// 	 FOR index := 1 TO GVL.gc_NumberStations DO
// 			GVL.g_Stations[index].P_eProcessMode := E_ProcessMode.Production;		   
// 	   END_FOR
// 		
// 	 
// 
// 	nExecutingSequence := nExecutingSequence +10;
// 
// 	10:
// 	  
// 	   
//   IF fbXPlanarMover[nTestID].P_Enable.Done THEN 
// 		stMoveOnTrackOptions.gap := 120;
// 		stMoveOnTrackOptions.direction := MC_DIRECTION.mcDirectionShortestWay;
// 		stMoveOnTrackOptions.dynamicMode := MC_DYNAMICS_REDUCTION_MODE.AccelerationLimitedVelocity;
// 
// 					
// 				fTargetPosOnTrack[1]:= GVL.g_Tracks[9].P_TrackLength;			
// 				fbXPlanarMover[nTestID].MoveOnTrackExt('move on track', GVL.g_Tracks[9].std, fTargetPosOnTrack[1],
// 								500, 2500, 50000, stMoveOnTrackOptions);
// 		nExecutingSequence := nExecutingSequence +1;
// 		 
// 	END_IF
// 
// 	11:
// 		bMoversInPos := TRUE;
// 		bMoverError := FALSE;
// 		
// 		
// 			bMoversInPos := bMoversInPos AND fbXPlanarMover[nTestID].P_MoveOnTrackExt.Done;
// 			bMoverError := bMoverError OR fbXPlanarMover[nTestID].P_MoveOnTrackExt.Error;
// 	
// 		
// 		IF bMoversInPos THEN
// 			nExecutingSequence := nExecutingSequence + 9;
// 		ELSIF bMoverError THEN
// 			nExecutingSequence := nExecutingSequence +  4;
// 		END_IF
// 
// 	20:
// 		FOR nForCounter:=1 TO GVL.gc_NumberStations DO
// 		IF GVL.g_Stations[nForCounter] <> 0 THEN
// 			GVL.g_Stations[nForCounter].Process();
// 			
// 			IF GVL.g_Stations[nForCounter].P_nErrorCode > 0 THEN
// 				nProcessFeedback := GVL.g_Stations[nForCounter].P_nErrorCode;
// 			END_IF
// 		END_IF
// 	END_FOR	
// 		nExecutingSequence := nExecutingSequence +10;
// 		
// 	30:
// 		stMoveOnTrackOptions.gap := 120;
// 		stMoveOnTrackOptions.direction := MC_DIRECTION.mcDirectionShortestWay;
// 		stMoveOnTrackOptions.dynamicMode := MC_DYNAMICS_REDUCTION_MODE.AccelerationLimitedVelocity;
// 		
// 		fTargetPosOnTrack[1] := GVL.g_Tracks[7].P_TrackLength;;
// 		fbXPlanarMover[nTestID].MoveOnTrackExt('move on track', GVL.g_Tracks[7].std, fTargetPosOnTrack[1],
// 												500, 2500, 50000, stMoveOnTrackOptions
// 		);
// 		nExecutingSequence := nExecutingSequence +1;
// 	31:
// 		// Movers moving on track
// 			bMoversInPos := TRUE;
// 			bMoverError := FALSE;
// 		
// 					bMoversInPos := bMoversInPos AND	fbXPlanarMover[nTestID].P_MoveOnTrackExt.Done;
// 					bMoverError := bMoverError OR fbXPlanarMover[nTestID].P_MoveOnTrackExt.Error;
// 	
// 			IF bMoversInPos THEN
// 			nExecutingSequence := nExecutingSequence + 9;
// 			ELSIF bMoverError THEN
// 			nExecutingSequence := nExecutingSequence + 4;
// 			END_IF
// 
// 
// 	40: 
// 
// 		stMoveOnTrackOptions.gap := 120;
// 		stMoveOnTrackOptions.direction := MC_DIRECTION.mcDirectionShortestWay;
// 		stMoveOnTrackOptions.dynamicMode := MC_DYNAMICS_REDUCTION_MODE.AccelerationLimitedVelocity;
// 		
// 		fTargetPosOnTrack[1] := GVL.g_Tracks[8].P_TrackLength;;
// 		fbXPlanarMover[nTestID].MoveOnTrackExt('move on track', GVL.g_Tracks[8].std, fTargetPosOnTrack[1],
// 												500, 2500, 50000, stMoveOnTrackOptions	);									
// 												
// 												
// 		nExecutingSequence := nExecutingSequence +1;
// 	41:
// 		// Movers moving on track
// 			bMoversInPos := TRUE;
// 			bMoverError := FALSE;
// 		
// 					bMoversInPos := bMoversInPos AND	fbXPlanarMover[nTestID].P_MoveOnTrackExt.Done;
// 					bMoverError := bMoverError OR fbXPlanarMover[nTestID].P_MoveOnTrackExt.Error;
// 	
// 			IF bMoversInPos THEN
// 			nExecutingSequence := nExecutingSequence + 9;
// 			ELSIF bMoverError THEN
// 			nExecutingSequence := nExecutingSequence + 4;
// 			END_IF
// 	
// 	
// 
// 	50:
// 		Execute := FALSE; // must be aborted manually
// 		nExecutingSequence := 0; // endless loop
	
END_CASE
END_METHOD

METHOD MoverPreparation : BOOL
VAR_INPUT
	bReset 	: BOOL;
END_VAR


VAR_INST
	
	nStatePreparation		: DINT;
	
	
	operationMode				: XPlanarOperationMode; 
	
	idx2						: UDINT;

	nTileDcLinkVoltage			: LREAL;
	bTilePowerOK				: BOOL;
	bTilePowerOverview			: ARRAY[1..GVL.gc_MaxNumberTiles] OF BOOL;
	bPowerOK					: BOOL;
	bPowerMissing				: BOOL;
	nTileCount					: UDINT;
	nTileToCheck				: UINT;
	bWithBumperID				: BOOL;	
	nMoverAccessoryIdCount		: ARRAY[1..GVL.gc_nMaxNumberMovers] OF UDINT;	
	
	stStartCheck 				: ST_CheckStartConditionFeedback;
	nLimitExceeded_MoverID		: UDINT;
	bLimitExceeded_Angle 		: BOOL;
	bLimitExceeded_PositionX 	: BOOL;
	bLimitExceeded_PositionY 	: BOOL;	
	fCurrentAngleDeviation		: LREAL;
	fCurrentPositionDeviationX	: LREAL;
	fCurrentPositionDeviationY	: LREAL;	

	sTextTemp					: STRING;

	eMoverAccessoryID			: MoverAccessoryID;

	
	moverCoordComStatus			: CoordinatedMoverCommStatus;
	moverComStatus				: MoverCommunicationStatus;
	
	bMoverCommunicationProblem  : ARRAY[1..GVL.gc_nMaxNumberMovers] OF BOOL;
	bCommunicationProblem		: BOOL;
	
	nMoverToCorrect				: UDINT;
	fMoverOrientationRead		: LREAL;
	fMoverOrientationCorrect	: LREAL;
	bDoRotationCorrection		: BOOL;
	CorrectionPos				: PositionXYC;
	
	bDeterminedMoverID				: BOOL;
	bDerterminedMoverOrientation 	: BOOL;
	
	fPosX							: LREAL;
	fPosY							: LREAL;
	fPosC							: LREAL;
	
	nCommunicationRetryCounter		: UINT;
	
	nMoverToCheck					: UINT;
	
	nMoverID_ErrorCode				: DWORD;
	
	MoverType						: XPlanarMoverType;
	bMoverCanDeterminOrientation	: BOOL;
	
			// Helper
	bDone 					: BOOL;
	idx						: UDINT;
	nForCounter 			: UDINT;	
	nErrorID				: UDINT;
	bMoverError				: BOOL;	
END_VAR
VAR
	sBtn: STRING(13);
END_VAR
IF bReset THEN
	nStatePreparation := 0;
	MoverPreparation := TRUE;
END_IF


	CASE nStatePreparation OF
		
	0:  nStatePreparation := 10;
	

	10: // 1st: Check if the system is in simulation mode or not
		// Simulation > OperationMode = 1
		//     Normal > OperationMode = 0
	    operationMode := fbXPlanarSystem.ipDriver.TcIoXpu(1).GetOperationMode();	
		IF operationMode = 0 THEN
			bPowerMissing := FALSE;
			nStatePreparation := nStatePreparation + 10;
		ELSE
			nStatePreparation := 500;
		END_IF
	
		
	20: // 2nd: Check power of each tile
		(*IF NOT bPowerMissing THEN
			ipVisuMessage.SetInfoMessage('Checking tile power', 'MoverPreparation', nStatePreparation);
		ELSE
			ipVisuMessage.SetErrorMessage('Tile power missing!', 'MoverPreparation', nStatePreparation, 0);	
		END_IF*)
		
		    bPowerOK := TRUE;
		nTileToCheck := 0;
		  nTileCount := fbXPlanarSystem.ipDriver.TcIoXpu(1).GetTileCount();
		
		nStatePreparation := nStatePreparation + 1;
		
	21:
		nTileToCheck := nTileToCheck +1;
		IF nTileToCheck <= nTileCount THEN
			nStatePreparation := nStatePreparation + 1;
		ELSE
			IF bPowerOK THEN
				nStatePreparation := nStatePreparation + 9;
			ELSE
				bPowerMissing := TRUE;
				nStatePreparation := nStatePreparation - 1;
			END_IF
		END_IF
		
	22:
		nTileDcLinkVoltage := fbXPlanarSystem.ipDriver.TcIoXpu(1).TcIoTile(1,nTileToCheck).GetDcLinkVoltage(); 
		IF nTileDcLinkVoltage > 6.0 THEN
			bTilePowerOK := TRUE;
		ELSE
			bTilePowerOK := FALSE;	
		END_IF
		bPowerOK := bPowerOK AND bTilePowerOK;
		bTilePowerOverview[nTileToCheck] := bPowerOK;
		nStatePreparation := nStatePreparation - 1;
		
		
		
	30:// 3rd: Mover re-detection, in case a mover was removed inbetween
	
		// Check if a mover has been lost...
		IF fbXPlanarSystem.CheckValidMovers() THEN
			//ipVisuMessage.SetInfoMessage('Mover re-detection', 'MoverPreparation', nStatePreparation);
		
		nStatePreparation := nStatePreparation + 1;
		END_IF
	
	31:
		IF fbXPlanarSystem.P_CheckValidMovers.bDone THEN
			IF fbXPlanarSystem.P_CheckValidMovers.bMoverLost THEN
				         bDeterminedMoverID := FALSE;
				bDerterminedMoverOrientation := FALSE;
				nStatePreparation := nStatePreparation + 1;
			ELSE
				nStatePreparation := nStatePreparation + 9;
			END_IF
		END_IF
				
		bDeterminedMoverID := FALSE;
		bDerterminedMoverOrientation := FALSE;		
		
		
	32: // Starting mover re-detection
		IF fbXPlanarSystem.UtilityCheckForError(bAutoReset := TRUE) > 0 THEN
			IF fbXPlanarSystem.ipDriver.TcIoXpu(1).SetStartMoverRedetection() THEN	
				nStatePreparation := nStatePreparation +1;
			END_IF
		END_IF
	
	33: // Checking if all movers have been found on the XPlanar surface
		stMoverDetectionInfos := fbXPlanarSystem.ipDriver.TcIoXpu(1).GetMoverDetectionInfos();
		gvl.g_nMoverCount := stMoverDetectionInfos.APM4220Detected ;
		
		
		IF stMoverDetectionInfos.APM4220Detected = stMoverDetectionInfos.APM4220Expected THEN
			nStatePreparation := nStatePreparation +7;
		ELSE
			sTextTemp := 'Mover Missing!  Expected:';
			sTextTemp := CONCAT(sTextTemp, UDINT_TO_STRING(stMoverDetectionInfos.APM4220Expected));
			sTextTemp := CONCAT(sTextTemp, '  Detected:');
			sTextTemp := CONCAT(sTextTemp, UDINT_TO_STRING(stMoverDetectionInfos.APM4220Detected));
			
			//ipVisuMessage.SetErrorMessage(sTextTemp, 'MoverPreparation', nStatePreparation, 0);	
		END_IF
	
	
	 40: // 4th: Checking the position of each mover before enabeling
	 	//ipVisuMessage.SetInfoMessage('Check mover position', 'MoverPreparation', nStatePreparation);
		stMoverDetectionInfos := fbXPlanarSystem.ipDriver.TcIoXpu(1).GetMoverDetectionInfos();	 	
		gvl.g_nMoverCount := stMoverDetectionInfos.APM4220Detected ;
		
		bDone := TRUE;
		FOR idx:=1 TO GVL.g_nMoverCount DO
			stStartCheck := GVL.g_Movers[idx].std.CheckStartConditions();
			IF NOT stStartCheck.bPositionOK THEN
				bDone := FALSE;
				EXIT;
			END_IF			
		END_FOR
	
		IF bDone THEN
			nStatePreparation := nStatePreparation + 2;
		ELSE
			nStatePreparation := nStatePreparation + 1;
		END_IF
			
	 41: // Position-Check failed:
		 // Except for rotation-points between four quadrants the angle limit of the c-axis is +/- 10.0°
		 // At rotation-points the max position deviation is +/-1mm in x/y-direction  	
				nLimitExceeded_MoverID := stStartCheck.nMoverID;
				  bLimitExceeded_Angle := stStartCheck.bAngleLimitExceeded;
			  bLimitExceeded_PositionX := stStartCheck.bPositionXLimitExceeded;
			  bLimitExceeded_PositionY := stStartCheck.bPositionYLimitExceeded;	
				fCurrentAngleDeviation := stStartCheck.fCurrentAngleDeviation;
			fCurrentPositionDeviationX := stStartCheck.fCurrentPositionDeviationX;
			fCurrentPositionDeviationY := stStartCheck.fCurrentPositionDeviationY;
	
			sTextTemp := 'Position Check Failed! - Mover ';
			sTextTemp := CONCAT(sTextTemp, UDINT_TO_STRING(nLimitExceeded_MoverID));
			sTextTemp := CONCAT(sTextTemp, ' too far away from rotation point.');
			
			//ipVisuMessage.SetErrorMessage(sTextTemp, 'MoverPreparation', nStatePreparation, 0);	
			
			nStatePreparation := nStatePreparation - 1;
			
	42:		//ipVisuMessage.ClearAllMessages();
			nStatePreparation := nStatePreparation + 8;
		
		
		
	50: // 5th: Check if movers with accessory MoverID are present. If yes, do mover identification before enabeling all movers.	
		bWithBumperID := FALSE;
			
		IF fbXPlanarSystem.UtilityCheckForError(bAutoReset := TRUE) > 0 THEN
			FOR idx:=1 TO GVL.g_nMoverCount DO
				nMoverAccessoryIdCount[idx] := fbXPlanarSystem.ipDriver.TcIoXpu(1).TcIoMover(UDINT_TO_UINT(idx)).GetMoverAccessoryIdCount();
			END_FOR
			
			FOR idx:=1 TO GVL.g_nMoverCount DO
				FOR idx2:=1 TO nMoverAccessoryIdCount[idx] DO
					eMoverAccessoryID := fbXPlanarSystem.ipDriver.TcIoXpu(1).TcIoMover(UDINT_TO_UINT(idx)).GetMoverAccessoryID(UDINT_TO_INT(idx2));
					
					IF eMoverAccessoryID = MoverAccessoryID.APM9001_0000 THEN
						// Note: With the current driver release (3.2209.36.0) mover identification only works if all movers are equiped with ID bumpers!
						bWithBumperID := TRUE;						
					END_IF
				END_FOR
			END_FOR
		END_IF

			
		IF bWithBumperID THEN
			nStatePreparation := nStatePreparation + 10;
		ELSE
			nStatePreparation := 500;
		END_IF
		
	
	60: // 6th: Do mover identification
		//ipVisuMessage.SetInfoMessage('Start mover-identification', 'MoverPreparation', nStatePreparation);
	
		IF NOT bDeterminedMoverID THEN
			IF fbXPlanarSystem.UtilityCheckForError(bAutoReset := TRUE) > 0 THEN
// 				IF fbXPlanarSystem.ipDriver.TcIoXpu(1).SetCoordMoverCommunicationCmd(CoordinatedMoverCommCommand.IdentifyAndAssignPossible) THEN
				IF fbXPlanarSystem.ipDriver.TcIoXpu(1).SetCoordMoverCommunicationCmd(CoordinatedMoverCommCommand.IdentifyBTNsAndRearrangeMovers) THEN
					nStatePreparation := nStatePreparation +1;
				END_IF	
			END_IF
		ELSE
			nStatePreparation := nStatePreparation +10;
		END_IF
	
	61:
		IF fbXPlanarSystem.UtilityCheckForError(bAutoReset := TRUE) > 0 THEN			
			moverCoordComStatus := fbXPlanarSystem.ipDriver.TcIoXpu(1).GetCoordMoverCommStatus();
			
			IF moverCoordComStatus = CoordinatedMoverCommStatus.CommunicationSuccessful THEN
				bDeterminedMoverID := TRUE;
				//ipVisuMessage.ClearAllMessages();
				nStatePreparation := nStatePreparation + 4;
			ELSIF moverCoordComStatus = CoordinatedMoverCommStatus.CommunicationFailed THEN
				nStatePreparation := nStatePreparation + 1;	
			END_IF
			
		END_IF
		
	62:	IF fbXPlanarSystem.UtilityCheckForError(bAutoReset := TRUE) > 0 THEN	
			nMoverID_ErrorCode := fbXPlanarSystem.ipDriver.TcIoXpu(1).GetCoordMoverCommunicationErrorId();
			//ipVisuMessage.SetErrorMessage('Mover Identification Failed!', 'MoverPreparation', nStatePreparation, nMoverID_ErrorCode);
		END_IF
		
		//IF ipVisuMessage.CheckAknowledge()  THEN
		nStatePreparation := 0;	
		//END_IF
	
	65: 
		FOR idx:=1 TO GVL.g_nMoverCount DO
			fbMover[idx].P_MoverID := fbXPlanarSystem.ipDriver.TcIoXpu(1).TcIoMover(UDINT_TO_UINT(idx)).GetIdentifiedMoverBtn();
		END_FOR
		nStatePreparation := nStatePreparation + 5;
	70: // 7th: Determine Mover-Orientation
	
		// Note: At the time of creation of this example code only APM4330 was able to determine its orientation.
		//       Change the code according to newer driver releases and availability of the orientation feature.
		bMoverCanDeterminOrientation := TRUE;
		FOR idx:=1 TO GVL.g_nMoverCount DO
			MoverType := fbXPlanarSystem.ipDriver.TcIoXpu(1).TcIoMover(UDINT_TO_UINT(idx)).GetMoverType();
			IF MoverType <> XPlanarMoverType.APM4330 THEN
				bMoverCanDeterminOrientation := FALSE;
			END_IF
		END_FOR
			
		IF bMoverCanDeterminOrientation THEN
			IF NOT bDerterminedMoverOrientation THEN
				//ipVisuMessage.SetInfoMessage('Mover orientation determination', 'MoverPreparation', nStatePreparation);
				IF fbXPlanarSystem.UtilityCheckForError(bAutoReset := TRUE) > 0 THEN
					IF fbXPlanarSystem.ipDriver.TcIoXpu(1).SetCoordMoverCommunicationCmd(CoordinatedMoverCommCommand.DetermineOrientations) THEN
						nStatePreparation := nStatePreparation + 1;	
					END_IF
				END_IF
			ELSE
				nStatePreparation := nStatePreparation + 20;		
			END_IF
		ELSE
			nStatePreparation := nStatePreparation + 20;
		END_IF
	
		
	71: // Check if communication is active
		IF fbXPlanarSystem.UtilityCheckForError(bAutoReset := TRUE) > 0 THEN
			moverCoordComStatus := fbXPlanarSystem.ipDriver.TcIoXpu(1).GetCoordMoverCommStatus();
			IF moverCoordComStatus = CoordinatedMoverCommStatus.CommunicationInProcess THEN
				nStatePreparation := nStatePreparation + 1;	
			END_IF
		END_IF
	
		
	72: // Wait for orientation determination finished
		IF fbXPlanarSystem.UtilityCheckForError(bAutoReset := TRUE) > 0 THEN
			moverCoordComStatus := fbXPlanarSystem.ipDriver.TcIoXpu(1).GetCoordMoverCommStatus();
			IF moverCoordComStatus = CoordinatedMoverCommStatus.CommunicationSuccessful THEN
				nStatePreparation := nStatePreparation + 8;	
			ELSIF moverCoordComStatus = CoordinatedMoverCommStatus.CommunicationFailed THEN
				IF nCommunicationRetryCounter <= 5 THEN
					nCommunicationRetryCounter := nCommunicationRetryCounter +1;
					nStatePreparation := nStatePreparation - 2;	
				ELSE
					nStatePreparation := nStatePreparation + 1;	
				END_IF
			END_IF
		END_IF
		
				
	73:	// Check which movers do not communicate correctly:
		nMoverToCheck := 0;
		nStatePreparation := nStatePreparation + 1;
		
	74: nMoverToCheck := nMoverToCheck +1;
		IF nMoverToCheck <= GVL.g_nMoverCount THEN
			IF fbXPlanarSystem.UtilityCheckForError(bAutoReset := TRUE) > 0 THEN
				IF fbXPlanarSystem.ipDriver.TcIoXpu(1).TcIoMover(nMoverToCheck).SetMoverCommunicationCommand(MoverCommunicationCommand.DetermineOrientation) THEN
					nStatePreparation := nStatePreparation + 1;
				END_IF
			END_IF
		ELSE
			FOR idx:=1 TO GVL.g_nMoverCount DO
				bCommunicationProblem := FALSE;
				IF bMoverCommunicationProblem[idx] THEN
					bCommunicationProblem := TRUE;	
				END_IF
			END_FOR
			
			IF bCommunicationProblem THEN
				sTextTemp := 'Mover Communication Problem: ';
				FOR idx:=1 TO GVL.g_nMoverCount DO
					IF bMoverCommunicationProblem[idx] THEN
						sTextTemp := CONCAT(sTextTemp, ' M');
						sTextTemp := CONCAT(sTextTemp, UDINT_TO_STRING(idx));
					END_IF
				END_FOR				
				//ipVisuMessage.SetErrorMessage(sTextTemp, sTextTemp, nStatePreparation, 0);
			ELSE
				nStatePreparation := nStatePreparation - 4;	
			END_IF
		END_IF
		
	75: moverComStatus := fbXPlanarSystem.ipDriver.TcIoXpu(1).TcIoMover(nMoverToCheck).GetCommunicationStatus();
		IF moverComStatus = MoverCommunicationStatus.CommunicationSuccessful THEN
			bMoverCommunicationProblem[nMoverToCheck] := FALSE;
			nStatePreparation := nStatePreparation - 1;
		ELSIF moverComStatus = MoverCommunicationStatus.CommunicationFailed THEN
			bMoverCommunicationProblem[nMoverToCheck] := TRUE;
			nStatePreparation := nStatePreparation - 1;
		END_IF
		
		
	80:	// Rotation-Angle modulo adaption
		//ipVisuMessage.SetInfoMessage('Rotation-Angle modulo adaption', 'MoverPreparation', nStatePreparation);
		nMoverToCorrect := 0;
		nStatePreparation := nStatePreparation + 1;	
		
	81:	nMoverToCorrect := nMoverToCorrect +1;
		IF nMoverToCorrect <= GVL.g_nMoverCount THEN
			fMoverOrientationRead    := GVL.g_Movers[nMoverToCorrect].std.P_ActPosition.c; 
			fMoverOrientationCorrect := fMoverOrientationRead;
			 bDoRotationCorrection := FALSE;
			nStatePreparation := nStatePreparation + 1;	
		ELSE
			bDerterminedMoverOrientation := TRUE;
			nStatePreparation := nStatePreparation + 9;	
		END_IF
		
	82:	IF fMoverOrientationCorrect >= 0 THEN
			IF fMoverOrientationCorrect > 360.0 THEN
				fMoverOrientationCorrect := fMoverOrientationCorrect - 180.0;
				bDoRotationCorrection := TRUE;
			ELSE
				nStatePreparation := nStatePreparation + 1;
			END_IF
		ELSE
			IF fMoverOrientationCorrect < 360.0 THEN
				fMoverOrientationCorrect := fMoverOrientationCorrect + 180.0;
				bDoRotationCorrection := TRUE;
			ELSE
				nStatePreparation := nStatePreparation + 1;
			END_IF
		END_IF			
		
		
	83:	IF bDoRotationCorrection THEN
			
			fPosX := GVL.g_Movers[nMoverToCorrect].std.P_ActPosition.x;
			fPosY := GVL.g_Movers[nMoverToCorrect].std.P_ActPosition.y;
			fPosC := GVL.g_Movers[nMoverToCorrect].std.P_ActPosition.c;
	
			CorrectionPos.SetValuesXYC(fPosX, fPosY, fMoverOrientationCorrect);	
	
			GVL.g_Movers[nMoverToCorrect].std.SetMoverPosition('Correction', CorrectionPos);
			
			nStatePreparation := nStatePreparation + 1;	
		ELSE
			nStatePreparation := nStatePreparation - 2;
		END_IF
		
	84:
		IF GVL.g_Movers[nMoverToCorrect].std.P_SetMoverPosition.Done THEN
			nStatePreparation := nStatePreparation - 3;
		ELSIF GVL.g_Movers[nMoverToCorrect].std.P_SetMoverPosition.Error THEN
			nErrorID := GVL.g_Movers[nMoverToCorrect].std.P_SetMoverPosition.ErrorID;
			//ipVisuMessage.SetErrorMessage('Rotation-Angle modulo adaption', 'MoverPreparation', nStatePreparation, nErrorID);
			GVL.g_Movers[nMoverToCorrect].P_ErrorID := UDINT_TO_INT(nErrorID);
			GVL.g_Movers[nMoverToCorrect].P_Error := TRUE;
		END_IF
		

	90: nStatePreparation := 500;
	
			
	500: // Done
	//	nStatePreparation := 0;
		MoverPreparation := TRUE;		
			
		
	END_CASE


	//ipVisuMessage.StateUpdate(nStatePreparation, 'MoverPreparation');
END_METHOD

METHOD MoverRecovery : BOOL
VAR_INPUT
	bReset : BOOL;
END_VAR

VAR
	index : UDINT;
	ipMoverApplication: INT;
END_VAR

VAR_INST
	
	stOptionsJoinTrack				: ST_JoinTrackOptions;
	bMoversJoined 					: BOOL;
	bMoverError 					: BOOL;
	bMoverOrientationSet			: BOOL;
	bClearStation 					:ARRAY [1..GVL.gc_NumberStations] OF BOOL;
	bStationCleared					:bool;
	nMoverToTurn					: UDINT;
	nMoverToTurnBack				: UDINT;
	nTrackToCheck					:UDINT; 
	nDistanceToTrack				:LREAL;
	nDistanceToTargetTrack			: ARRAY[1..moverCount] OF REAL;
	nTargetTrack					: ARRAY[1..moverCount] OF UDINT;
	
	
	
	fRecoveryRotTarget				: LREAL;
	fRecoveryRotVel					: LREAL :=  360.0;
	fRecoveryRotAcc					: LREAL := 1800.0;
	fRecoveryRotJerk				: LREAL := 9000.0;
	stRotationOptions				: ST_MoveCOptions;




	
END_VAR
IF bReset THEN
	MoverRecovery := FALSE;
	nRecoverySequence := 0;
END_IF

CASE nRecoverySequence OF
	0:
		bMoversJoined := FALSE;
		bMoverError := FALSE;
		nMoverToTurn := 0;
		IF NOT bReset THEN
			nRecoverySequence := nRecoverySequence + 1;
		END_IF
		
	1: 	//set rotary orienation 
	
		FOR index := 1 TO gvl.g_nMoverCount DO
		fbXPlanarMover[index].MoveA('', 0, 100, 1000, 1000, 10000);
		fbXPlanarMover[index].MoveB('', 0, 100, 1000, 1000, 10000);
 		fbXPlanarMover[index].MoveC('', 0, 180, 1800, 1800, 18000, 0);
		
		END_FOR

		nRecoverySequence := nRecoverySequence + 1;
	
	2: 
		bMoverOrientationSet:= TRUE; 
		FOR index := 1 TO  gvl.g_nMoverCount DO
			IF fbXPlanarMover[index].P_MoveA.Done AND fbXPlanarMover[index].P_MoveB.Done AND fbXPlanarMover[index].P_MoveC.Done THEN 
				bMoverOrientationSet:= TRUE; 
			ELSE 
				bMoverOrientationSet:= FALSE; 
				
			END_IF
		END_FOR
		
		IF bMoverOrientationSet THEN
			nRecoverySequence := nRecoverySequence + 8;
	
		END_IF
	
	10:
	
		nMoverToTurn := nMoverToTurn +1;
		IF nMoverToTurn > gvl.g_nMoverCount THEN
				nRecoverySequence := nRecoverySequence +3;
			ELSE
				IF GVL.g_Movers[nMoverToTurn].std.P_IsPresent THEN

					fRecoveryRotTarget 				  := GVL.g_Movers[nMoverToTurn].std.P_ClosestQuaterAngle;	
					stRotationOptions.additionalTurns := 0;
					stRotationOptions.direction		  := Tc3_Mc3PlanarMotion.MC_direction.mcDirectionNonModulo;	
					
					GVL.g_Movers[nMoverToTurn].std.MoveC('Recovery - unfinished rotation', fRecoveryRotTarget, fRecoveryRotVel, fRecoveryRotAcc, fRecoveryRotAcc, fRecoveryRotJerk, stRotationOptions);
					nRecoverySequence := nRecoverySequence +1;				
				END_IF	
			END_IF
		
	
	11:
			IF GVL.g_Movers[nMoverToTurn].std.P_MoveC.Done THEN
				nRecoverySequence := nRecoverySequence -1;	
			ELSIF GVL.g_Movers[nMoverToTurn].std.P_MoveC.Error THEN
				nRecoverySequence := nRecoverySequence +1;	
			END_IF
			
	12: 		// Check error ID and react accordingly
			nErrorID := GVL.g_Movers[nMoverToTurn].std.P_MoveC.ErrorID;
			GVL.g_Movers[nMoverToTurn].P_ErrorID := UDINT_TO_INT(nErrorID);
			GVL.g_Movers[nMoverToTurn].P_Error := TRUE;

			// In case rotation is not possible due to collision with another mover proceed without rotation correction.
			IF nErrorID = 33158 THEN
				nRecoverySequence := nRecoverySequence -2;
			END_IF

	13: 	nRecoverySequence := 100;	

		    
	100: 
			bStationCleared:=TRUE;
			bClearStation[GVL.PuncherStation]:=fbPuncherStation.Clear();
			bClearStation[GVL.PuncherSeparateStation]:=fbPuncherSeparateStation.Clear();
			bClearStation[GVL.PuncherBufferStation]:=fbPuncherBufferStation.Clear();
	
	FOR  index := 1 TO  GVL.gc_NumberStations DO
		IF bClearStation[index] THEN
			bStationCleared:=TRUE;
			ELSE
				bStationCleared:=FALSE;
		END_IF
	END_FOR
	IF bStationCleared THEN
			nRecoverySequence := 200;

		END_IF
		
// 	110: // look for for nearest track 
// 	
// 	
// 	FOR nMoverToTurnBack := 1 TO  gvl.g_nMoverCount DO
// 		nDistanceToTargetTrack[nMoverToTurnBack]:= 999999;
// 		
// 		FOR nTrackToCheck :=1 TO GVL.gc_NumberTracks DO 
// 		nDistanceToTrack := fbXPlanarMover[ nMoverToTurnBack].GetDistanceToTrack(GVL.g_Tracks[nTrackToCheck].std);
// 		
// 		IF nDistanceToTrack < nDistanceToTargetTrack[nMoverToTurnBack] AND nDistanceToTrack<> -1 THEN 
// 			nDistanceToTargetTrack[nMoverToTurnBack]:=nDistanceToTrack;
// 			nTargetTrack[nMoverToTurnBack] :=nTrackToCheck;
// 		END_IF
// 		
// 	END_FOR
// 	
// 	END_FOR
// 	
// 	nRecoverySequence := nRecoverySequence +10;
// 	
// 	120: // join to track
// 
// 		stOptionsJoinTrack.useOrientation := TRUE;
// 		
// 		FOR index := 1 TO gvl.g_nMoverCount DO
// 		IF fbXPlanarMover[index].P_CommandMode<> MC_PLANAR_MOVER_COMMAND_MODE.OnTrack THEN
// 			fbXPlanarMover[index].JoinTrack('Joining track', GVL.g_Tracks[nTargetTrack[index]].std, 250, 1250, 12500, stOptionsJoinTrack);
// 			
// 		END_IF
// 		
// 			
// END_FOR
// 	
// 		nRecoverySequence := nRecoverySequence + 1;
// 		
// 	121:
// 		bMoversJoined := TRUE;
// 		bMoverError := FALSE;
// 		FOR index := 1 TO moverCount DO
// 			bMoversJoined := bMoversJoined AND fbXPlanarMover[index].P_JoinTrack.Done;
// 			IF  fbXPlanarMover[index].P_JoinTrack.Done THEN 
// 				gvl.g_Movers[index].P_TrackId:=nTargetTrack[index];
// 			END_IF
// 			bMoverError := bMoverError OR fbXPlanarMover[index].P_JoinTrack.Error;			
// 		END_FOR
// 		
// 	IF bMoversJoined THEN
// 			nRecoverySequence := nRecoverySequence + 9;
// 	ELSIF bMoverError THEN
//  			nRecoverySequence := nRecoverySequence + 4;
// 	END_IF
// 		
		
// 	130: //send mover to station 
// 	  	  
// 		FOR index := 1 TO gvl.g_nMoverCount DO
// 			 IF fbXPlanarMover[index].P_TrackId= GVL.TrackPuncherWellplate THEN 
// 				 fbPuncherStation.P_List_Switch_Input_W.AddMover(GVL.g_Movers[index].std);
// 		
// 			
// 			 END_IF
// 		END_FOR
// 
// 		nRecoverySequence := 200;

	200: 
		MoverRecovery := TRUE;
		
END_CASE
END_METHOD

METHOD Resetting : BOOL
VAR_INPUT
END_VAR

VAR
	index : UDINT;
	MC_PLANNAR_: ST_CommandReturn;
END_VAR


VAR_INST
	
	nTrackToEnable		: UDINT;
	stProductDataClear 	: ST_ProductData;
	stOptionsJoinTrack				: ST_JoinTrackOptions;
	bMoversJoined 					: BOOL;
	bMoverError 					: BOOL;
	nMoverToTurn					: UDINT;
	nMoverToTurnBack				: UDINT;
	nTrackToCheck					:UDINT; 
	nDistanceToTrack				:LREAL;
	nDistanceToTargetTrack			: ARRAY[1..moverCount] OF REAL;
	nTargetTrack					: ARRAY[1..moverCount] OF UDINT;
	
END_VAR
nErrorID := 0;

CASE nResettingSequence OF 
	
	0: // Enter 
		nResettingSequence := 10;
		
		
		
	10: // Reset all movers
		IF fbXPlanarSystem.ResetMovers() THEN
		//	ipVisuMessage.SetInfoMessage('RESET all movers', 'Resetting', nResettingSequence);
			nResettingSequence := nResettingSequence +1;			
		END_IF
		
	11: IF fbXPlanarSystem.P_ResetMovers.Done THEN
			nResettingSequence := nResettingSequence +9;
		ELSIF fbXPlanarSystem.P_ResetMovers.Error THEN
			nResettingSequence := nResettingSequence +1;	
		END_IF

	12:	// Check error ID and react accordingly
		nErrorID := fbXPlanarSystem.P_EnableMovers.ErrorID;
		//ipVisuMessage.SetErrorMessage('RESET movers failed', 'Resetting', nResettingSequence, nErrorID);					
		
		
		
	20:	// Reset all tracks
		IF fbXPlanarSystem.ResetTracks() THEN
			//ipVisuMessage.SetInfoMessage('RESET all tracks', 'Resetting', nResettingSequence);
			nResettingSequence := nResettingSequence +1;
		END_IF
		
	21: IF fbXPlanarSystem.P_ResetTracks.Done THEN
			nResettingSequence := nResettingSequence +19;
	 	ELSIF fbXPlanarSystem.P_ResetTracks.Error THEN
			nResettingSequence := nResettingSequence +1;	
		END_IF
	
	22:	// Check error ID and react accordingly
		nErrorID := fbXPlanarSystem.P_EnableMovers.ErrorID;
		//ipVisuMessage.SetErrorMessage('RESET tracks failed', 'Resetting', nResettingSequence, nErrorID);			
		
	
		
// 	30:	// Reset MotionSystemApplication
// 		IF ipMotionSystemApplication.Reset() THEN
// 		//	ipVisuMessage.SetInfoMessage('RESET MotionSystemApplication', 'Resetting', nResettingSequence);
// 			nResettingSequence := nResettingSequence +10;
// 		END_IF
	
				
	40:  // Cleaning all process data
		FOR idx:=1 TO GVL.g_nMoverCount DO
		//	ipMoverApplication[idx].P_ProductData := stProductDataClear;
		END_FOR
		nResettingSequence := nResettingSequence+10;
		
	50: // check if any mover is disable 
			
		FOR index := 1 TO gvl.g_nMoverCount DO
			 IF fbXPlanarMover[index].P_State=MC_PLANAR_STATE.Disabled THEN 
				 nResettingSequence := nResettingSequence + 1;
				 RETURN; 
			 END_IF
		END_FOR
			 nResettingSequence :=100;
	 
	51:	// enable movers
			IF fbXPlanarSystem.EnableMovers() THEN
				nResettingSequence := nResettingSequence + 1;
			END_IF
	
	52: // wait for enabling
		IF fbXPlanarSystem.P_EnableMovers.Done THEN
			nResettingSequence := 100;
		ELSIF fbXPlanarSystem.P_EnableMovers.Error THEN
			nResettingSequence := nResettingSequence + 3;
			nErrorID := fbXPlanarSystem.P_EnableMovers.ErrorID;
 		END_IF
		
// 	60:  // look for for nearest track 
// 	
// 		FOR nMoverToTurnBack := 1 TO  gvl.g_nMoverCount DO
// 			nDistanceToTargetTrack[nMoverToTurnBack]:= 999999;
// 			
// 			FOR nTrackToCheck :=1 TO 10 DO//GVL.gc_NumberTracks DO 
// 			nDistanceToTrack := fbXPlanarMover[ nMoverToTurnBack].GetDistanceToTrack(GVL.g_Tracks[nTrackToCheck].std);
// 			
// 				IF nDistanceToTrack < nDistanceToTargetTrack[nMoverToTurnBack] THEN 
// 					nDistanceToTargetTrack[nMoverToTurnBack]:=nDistanceToTrack;
// 					nTargetTrack[nMoverToTurnBack] :=nTrackToCheck;
// 				END_IF
// 			
// 			END_FOR
// 	
// 		END_FOR
// 		
// 	nResettingSequence := nResettingSequence +10;
// 	
// 	70: // join to track
// 
// 		stOptionsJoinTrack.useOrientation := TRUE;
// 		
// 		FOR index := 1 TO gvl.g_nMoverCount DO
// 		IF fbXPlanarMover[index].P_CommandMode<> MC_PLANAR_MOVER_COMMAND_MODE.OnTrack THEN
// 			fbXPlanarMover[index].JoinTrack('Joining track', GVL.g_Tracks[nTargetTrack[index]].std, 250, 1250, 12500, stOptionsJoinTrack);
// 			END_IF
// 
// END_FOR
// 	
// 		nResettingSequence := nResettingSequence + 1;
// 		
// 	71:
// 		bMoversJoined := TRUE;
// 		bMoverError := FALSE;
// 		FOR index := 1 TO moverCount DO
// 			bMoversJoined := bMoversJoined AND fbXPlanarMover[index].P_JoinTrack.Done;
// 			bMoverError := bMoverError OR fbXPlanarMover[index].P_JoinTrack.Error;			
// 		END_FOR
// 		
// 	IF bMoversJoined THEN
// 			nResettingSequence := 100;
// 	ELSIF bMoverError THEN
//  			nResettingSequence := nResettingSequence + 4;
// 	END_IF
// 		
	
	100: // Reset done
		//ipVisuMessage.SetInfoMessage('RESET finished', 'Resetting', 0);
	
		nResettingSequence := 0; 
		         Resetting := TRUE;

END_CASE



//ipVisuMessage.StateUpdate(nResettingSequence, 'Resetting');
END_METHOD

METHOD Starting : BOOL
VAR_INPUT
	bReset : BOOL;
END_VAR

VAR 
	nErrorID : UDINT;
	nMoverIndex: UDINT;
END_VAR
IF bReset THEN
	Starting := FALSE;
	nStartingSequence := 0;
END_IF

CASE nStartingSequence OF
	0: //init
		Execute(bReset := TRUE);
		MoverRecovery(bReset := TRUE);
		IF NOT bReset THEN
			nStartingSequence := nStartingSequence + 10;
		END_IF
	10: // enable collision avoidance group
		IF fbXPlanarSystem.EnableGroup() THEN
			nStartingSequence := nStartingSequence + 1;
		END_IF
	11:
		IF fbXPlanarSystem.P_EnableGroup.Done THEN
			nStartingSequence := nStartingSequence + 9;
		ELSIF fbXPlanarSystem.P_EnableGroup.Error THEN
			nStartingSequence := nStartingSequence + 4;
			nErrorID := fbXPlanarSystem.P_EnableGroup.ErrorID;
		END_IF
	20: // add environment 
		IF fbXPlanarSystem.AddEnvironmentToGroup() THEN
			nStartingSequence := nStartingSequence + 1;
		END_IF
	21: 
		IF fbXPlanarSystem.P_AddEnviromentToGroup.Done THEN
			nStartingSequence := nStartingSequence + 9;
		ELSIF fbXPlanarSystem.P_AddEnviromentToGroup.Error THEN
			nStartingSequence := nStartingSequence + 4;
			nErrorID := fbXPlanarSystem.P_AddEnviromentToGroup.ErrorID;
		END_IF
		
	30:
		IF fbXPlanarSystem.EnableTracks() THEN
			nStartingSequence := nStartingSequence + 1;
		END_IF
	
	31: 
		IF fbXPlanarSystem.P_EnableTracks.Done THEN
			nStartingSequence := nStartingSequence + 9;
		ELSIF fbXPlanarSystem.P_EnableTracks.Error THEN
			nStartingSequence := nStartingSequence + 4;
			nErrorID := fbXPlanarSystem.P_EnableTracks.ErrorID;
		END_IF
	
			
	40:
		IF fbXPlanarSystem.AddTracksToGroup() THEN
			nStartingSequence := nStartingSequence + 1;
		END_IF
	
	41: 
		IF fbXPlanarSystem.P_AddTracksToGroup.Done THEN
			nStartingSequence := nStartingSequence + 1;
		ELSIF fbXPlanarSystem.P_AddTracksToGroup.Error THEN
			nStartingSequence := nStartingSequence + 4;
			nErrorID := fbXPlanarSystem.P_AddTracksToGroup.ErrorID;
		END_IF
		
	42: // Prepare all movers
		IF MoverPreparation(bReset:=TRUE) THEN
			nStartingSequence := nStartingSequence + 1;
		END_IF
		
	43:
		IF MoverPreparation(bReset:=FALSE) THEN
			nStartingSequence := nStartingSequence + 7;
		END_IF	
		
	50: // enable movers
		IF fbXPlanarSystem.EnableMovers() THEN
			nStartingSequence := nStartingSequence + 1;
		END_IF
	51: // wait for enabling
		IF fbXPlanarSystem.P_EnableMovers.Done THEN
			nStartingSequence := nStartingSequence + 9;
		ELSIF fbXPlanarSystem.P_EnableMovers.Error THEN
			nStartingSequence := nStartingSequence + 4;
			nErrorID := fbXPlanarSystem.P_EnableMovers.ErrorID;
		END_IF
	60: // add movers to group
		IF fbXPlanarSystem.AddMoversToGroup() THEN
			nStartingSequence := nStartingSequence + 1;
		END_IF
	61: // wait for enabling
		IF fbXPlanarSystem.P_AddMoversToGroup.Done THEN
			nStartingSequence := nStartingSequence + 1;
		ELSIF fbXPlanarSystem.P_AddMoversToGroup.Error THEN
			nStartingSequence := nStartingSequence + 4;
			nErrorID := fbXPlanarSystem.P_AddMoversToGroup.ErrorID;
		END_IF
	62:
	 	FOR nMoverIndex := 1 TO GVL.g_nMoverCount DO
			GVL.g_Movers[nMoverIndex].std.P_Id := UDINT_TO_UINT(nMoverIndex);
		END_FOR
		nStartingSequence := nStartingSequence + 8;
	70:
		IF MoverRecovery(bReset := FALSE) THEN
			nStartingSequence := nStartingSequence + 10;
		END_IF
	80: 
		Starting := TRUE;
END_CASE
END_METHOD

METHOD Startup : BOOL
VAR_INPUT
	bReset : BOOL;
END_VAR

VAR
	index : UDINT;
		stMoverDetectionInfos   : ST_TcIoMoverDetectionInfos;
		detectedMovers:UDINT;
END_VAR

VAR_INST
	aTrackTable : ARRAY[1..maxTrackCount] OF FB_TrackTable;
	nTrackIdx: UDINT;
	nStationToInit : UINT;
	
	nStartFromTrack : UDINT;
	nEndAtTrack : UDINT;
	bCloseLoop : BOOL;
END_VAR
IF bReset THEN
	Startup := FALSE;
	nStartupSequence := 0;
END_IF

CASE nStartupSequence OF
	0: //init
		bAssignmentComplete := FALSE;
		IF NOT bReset THEN
			nStartupSequence := nStartupSequence + 1;
		END_IF

	1: //assign mover to system
		
		FOR index := 1 TO MoverCount DO
			fbMover[index].std := THIS^.fbXPlanarMover[index];
		END_FOR	
		//nStartupSequence := nStartupSequence + 1;
	
		FOR index := 1 TO moverCount DO
			fbXPlanarSystem.SetMoverStandard(index, THIS^.fbXPlanarMover[index]);
		END_FOR
		
		nStartupSequence := nStartupSequence + 1;
		
	2:  // Movers to global mover interface
		FOR index := 1 TO MoverCount DO
			GVL.g_Movers[index] := THIS^.fbMover[index];
			THIS^.fbMover[index].P_MoverIndex := UDINT_TO_INT(index); 
		END_FOR	
		nStartupSequence := nStartupSequence + 1;
	
	3:  // Assigning global Track-Interfaces
		GVL.g_Tracks[GVL.TrackPuncherWellplate] := THIS^.fbTrackPuncherWellplate;
		GVL.g_Tracks[GVL.TrackBufferPuncher] := THIS^.fbTrackBufferPuncher;
		GVL.g_Tracks[GVL.TrackStradeFirstSeg] := THIS^.fbTrackStradeFirstSeg;
		GVL.g_Tracks[GVL.TrackStradeSecondSeg] := THIS^.fbTrackStradeSecondSeg;
		GVL.g_Tracks[GVL.TrackPipettePreBuffer] := THIS^.fbTrackPipettePreBuffer;
		GVL.g_Tracks[GVL.TrackPipette] := THIS^.fbTrackPipette;
		GVL.g_Tracks[GVL.TrackPipettePostBuffer] := THIS^.fbTrackPipettePostBuffer;
		GVL.g_Tracks[GVL.TrackPipetteBufferCon] := THIS^.fbTrackPipetteBufferCon;
		GVL.g_Tracks[GVL.TrackUserInteraction] := THIS^.fbTrackUserInteraction;
		GVL.g_Tracks[GVL.CloseLoopTrack] := THIS^.fbCloseLoopTrack;
		GVL.g_Tracks[GVL.PuncherSeperateTrack] := THIS^.fbPuncherSeperate;
		
		
		nTrackIdx := 0;
		bAssignmentComplete := TRUE;
		nStartupSequence := nStartupSequence + 1;	
		
	4: //assign track to system
		FOR index := 1 TO GVL.gc_NumberTracks DO
			fbXPlanarSystem.SetTrackStandard(index, GVL.g_Tracks[index].std);
		END_FOR
		
		nStartupSequence := nStartupSequence + 1;
	
	5: // assign stations
		GVL.g_Stations[GVL.PuncherStation] := THIS^.fbPuncherStation;
		GVL.g_Stations[GVL.PuncherSeparateStation] := THIS^.fbPuncherSeparateStation;
		GVL.g_Stations[GVL.PuncherBufferStation] := THIS^.fbPuncherBufferStation;
		
		nStartupSequence := nStartupSequence + 6;
		
	11: // Track number count
		IF nTrackIdx < GVL.gc_NumberTracks THEN
			nTrackIdx := nTrackIdx + 1;
			nStartupSequence := nStartupSequence +1;
		ELSE
			    nTrackIdx := 0;
			nStartupSequence := 14;
		END_IF
				
	12:	// Clear track data
		IF GVL.g_Tracks[nTrackIdx].Clear() THEN
			nStartupSequence := nStartupSequence +1;
		END_IF
		
	13: // Build the track
		IF GVL.g_Tracks[nTrackIdx].Initialize(nTrackIdx) THEN	
			nStartupSequence := 11;
		ELSE
			IF GVL.g_Tracks[nTrackIdx].P_Error THEN
				nStartupSequence := nStartupSequence +1;
			END_IF
		END_IF
		
	14: // Init all stations
		nStationToInit := 0;
		nStartupSequence := nStartupSequence +1;

	15:	nStationToInit := nStationToInit +1;
		IF nStationToInit <= GVL.gc_NumberStations THEN
			nStartupSequence := nStartupSequence +1;
		ELSE
			nStartupSequence := 30;
		END_IF	
				
	16: IF GVL.g_Stations[nStationToInit].Init() THEN
			nStartupSequence := nStartupSequence -1;
		END_IF

	30: 
		Startup := TRUE;
END_CASE
END_METHOD

END_FUNCTION_BLOCK

// ---- Tracks/FB_PuncherBufferTrack.TcPOU
FUNCTION_BLOCK FB_PuncherBufferTrack EXTENDS FB_BaseTrack implements I_Track;
VAR_INPUT
END_VAR
VAR_OUTPUT
END_VAR
VAR
END_VAR

METHOD Initialize : BOOL
VAR_INPUT
	nTrackIndex	: UDINT;
END_VAR

VAR_INST
	TrackTable		: FB_TrackTable;
	
END_VAR


CASE nInitState OF
	10:	// Starting with an empty table. 
		IF TrackTable.ClearTrackTable() THEN
			nInitState := nInitState + 10;
		END_IF
	20: 
		// Init Track-Table
		
		// *************************************************************************************
		// *** Only the code in this state must be eddited according to machine/track layout ***
		// *************************************************************************************	
		
		nStartFromTrack	:= 1;		// 0 for the first track all others according to their predecessor!
	    	nEndAtTrack := 0;		// 0 for the first track all others according to their successor! 		
		     bCloseLoop := FALSE;	// TRUE for circular track	
		
		TrackTable.AddPoint(E_PointType.Line_Start, E_PointOption.none, 540, 310, 0);
		TrackTable.AddPoint(E_PointType.Line_End, E_PointOption.none, 540, 410, 0);
			 
			 
		TrackTable.AddPoint(E_PointType.Line_Start, E_PointOption.none, 550, 420, 0);
		TrackTable.AddPoint(E_PointType.Line_End, E_PointOption.none, 660, 420, 0);
		
		nInitState := nInitState + 10;
		
	30:
		// *************************************************************
		// ***       NO Code Changes are needed from here on!        ***
		// *************************************************************		
			
		// The track table contains all additional information, too.
		IF nStartFromTrack > 0 THEN
			TrackTable.P_StartFromTrack := GVL.g_Tracks[nStartFromTrack].std;	
		END_IF
		IF nEndAtTrack > 0 THEN
			TrackTable.P_EndAtTrack := GVL.g_Tracks[nEndAtTrack].std;	
		END_IF	
		TrackTable.P_CloseTheLoop := bCloseLoop;	
		nInitState := nInitState + 10;

			
		
	40: // Checking the track table for plausibility
		IF TrackTable.CheckTrackTable() <> 0 THEN
			IF TrackTable.P_TrackTableCheckResult THEN
				nInitState := 50;	// Plausibility test succeeded.
			ELSE
				nInitState := 41;	// Plausibility test failed!
			END_IF
		END_IF
	41:	// In case of failed plausibility test check the creation of the above track table.
		// A Line must always begin with E_PointType.Line_Start and end with E_PointType.Line_End.
		// A Circle must always be added in the order E_PointType.Circle_Start, E_PointType.Circle_Center, E_PointType.Circle_End.
		// Check the info text for further information:
		bTrackBuildError := TRUE;
							
 					   
	50:	// Building the track	
		IF fbTrackStandard.BuildTrackExt(TrackTable) THEN
			nInitState := nInitState +1;
		END_IF
		
	51:	IF fbTrackStandard.P_BuildTrackExt.Done THEN
			nInitState := 100;	
		ELSIF fbTrackStandard.P_BuildTrackExt.Error THEN
	  		nInitState := nInitState +1;
		END_IF		
		
	52: // In case an error occured, check the error ID and InfoText and react accordingly:
		   bTrackBuildError := TRUE;
		 
	100: 	// Track build done
			fTrackLength := fbTrackStandard.GetLength();
			  Initialize := TRUE;
	
			
END_CASE
END_METHOD

PROPERTY P_Error : Bool
GET
P_Error := bTrackBuildError;
END_GET
END_PROPERTY

END_FUNCTION_BLOCK

// ---- Tracks/FB_PipetteTrack.TcPOU
FUNCTION_BLOCK FB_PipetteTrack EXTENDS FB_BaseTrack implements I_Track;
VAR_INPUT
END_VAR
VAR_OUTPUT
END_VAR
VAR
END_VAR

METHOD Initialize : BOOL
VAR_INPUT
	nTrackIndex	: UDINT;
END_VAR

VAR_INST
	TrackTable		: FB_TrackTable;
	
	bIsDone : BOOL;
	bIsActive : BOOL;
	bIsError : BOOL;
	stRet : ST_CommandReturn;
END_VAR


CASE nInitState OF
	10:	// Starting with an empty table. 
		IF TrackTable.ClearTrackTable() THEN
			nInitState := nInitState + 10;
		END_IF
	20: 
		// Init Track-Table
		
		// *************************************************************************************
		// *** Only the code in this state must be eddited according to machine/track layout ***
		// *************************************************************************************	
		
		nStartFromTrack	:= 5;		// 0 for the first track all others according to their predecessor!
	    	nEndAtTrack := 0;		// 0 for the first track all others according to their successor! 		
		     bCloseLoop := FALSE;	// TRUE for circular track	
		
		TrackTable.AddPoint(E_PointType.Line_Start, E_PointOption.none, 180, 299.99, 0);
		TrackTable.AddPoint(E_PointType.Line_End, E_PointOption.none, 180, 60.01, 0);
		
		TrackTable.AddPoint(E_PointType.Line_Start, E_PointOption.none, 179.99, 60, 0);
		TrackTable.AddPoint(E_PointType.Line_End, E_PointOption.none, 120, 60, 0);
		nInitState := nInitState + 10;
		
	30:
		// *************************************************************
		// ***       NO Code Changes are needed from here on!        ***
		// *************************************************************		
			
		// The track table contains all additional information, too.
		IF nStartFromTrack > 0 THEN
			TrackTable.P_StartFromTrack := GVL.g_Tracks[nStartFromTrack].std;	
		END_IF
		IF nEndAtTrack > 0 THEN
			TrackTable.P_EndAtTrack := GVL.g_Tracks[nEndAtTrack].std;	
		END_IF	
		TrackTable.P_CloseTheLoop := bCloseLoop;	
		nInitState := nInitState + 10;

			
		
	40: // Checking the track table for plausibility
		IF TrackTable.CheckTrackTable() <> 0 THEN
			IF TrackTable.P_TrackTableCheckResult THEN
				nInitState := 50;	// Plausibility test succeeded.
			ELSE
				nInitState := 41;	// Plausibility test failed!
			END_IF
		END_IF
	41:	// In case of failed plausibility test check the creation of the above track table.
		// A Line must always begin with E_PointType.Line_Start and end with E_PointType.Line_End.
		// A Circle must always be added in the order E_PointType.Circle_Start, E_PointType.Circle_Center, E_PointType.Circle_End.
		// Check the info text for further information:
		bTrackBuildError := TRUE;
							
 					   
	50:	// Building the track	
		IF fbTrackStandard.BuildTrackExt(TrackTable) THEN
			nInitState := nInitState +1;
		END_IF
		
	51:	
		bIsDone := fbTrackStandard.P_BuildTrackExt.Done;
		bIsActive := fbTrackStandard.P_BuildTrackExt.Active;
		bIsError := fbTrackStandard.P_BuildTrackExt.Error;
		stRet := fbTrackStandard.P_BuildTrackExt;
		
		IF fbTrackStandard.P_BuildTrackExt.Done THEN
			nInitState := 100;	
		ELSIF fbTrackStandard.P_BuildTrackExt.Error THEN
	  		nInitState := nInitState +1;
		END_IF		
		
	52: // In case an error occured, check the error ID and InfoText and react accordingly:
		   bTrackBuildError := TRUE;
		 
	100: 	// Track build done
			fTrackLength := fbTrackStandard.GetLength();
			  Initialize := TRUE;
	
			
END_CASE
END_METHOD

PROPERTY P_Error : Bool
GET
P_Error := bTrackBuildError;
END_GET
END_PROPERTY

END_FUNCTION_BLOCK

// ---- Tracks/FB_CloseLoopTrack.TcPOU
FUNCTION_BLOCK FB_CloseLoopTrack EXTENDS FB_BaseTrack implements I_Track;
VAR_INPUT
END_VAR
VAR_OUTPUT
END_VAR
VAR
END_VAR

METHOD Initialize : BOOL
VAR_INPUT
	nTrackIndex	: UDINT;
END_VAR

VAR_INST
	TrackTable		: FB_TrackTable;
	
	bIsDone : BOOL;
	bIsActive : BOOL;
	bIsError : BOOL;
	stRet : ST_CommandReturn;
END_VAR


CASE nInitState OF
	10:	// Starting with an empty table. 
		IF TrackTable.ClearTrackTable() THEN
			nInitState := nInitState + 10;
		END_IF
	20: 
		// Init Track-Table
		
		// *************************************************************************************
		// *** Only the code in this state must be eddited according to machine/track layout ***
		// *************************************************************************************	
		
		nStartFromTrack	:= 9;		// 0 for the first track all others according to their predecessor!
	    	nEndAtTrack := 0;		// 0 for the first track all others according to their successor! 		
		     bCloseLoop := FALSE;	// TRUE for circular track	
		
		TrackTable.AddPoint(E_PointType.Line_Start, E_PointOption.none, 190, 420, 0);
		TrackTable.AddPoint(E_PointType.Line_End, E_PointOption.none, 530, 420, 0);
		
		
		nInitState := nInitState + 10;
		
	30:
		// *************************************************************
		// ***       NO Code Changes are needed from here on!        ***
		// *************************************************************		
			
		// The track table contains all additional information, too.
		IF nStartFromTrack > 0 THEN
			TrackTable.P_StartFromTrack := GVL.g_Tracks[nStartFromTrack].std;	
		END_IF
		IF nEndAtTrack > 0 THEN
			TrackTable.P_EndAtTrack := GVL.g_Tracks[nEndAtTrack].std;	
		END_IF	
		TrackTable.P_CloseTheLoop := bCloseLoop;	
		nInitState := nInitState + 10;

			
		
	40: // Checking the track table for plausibility
		IF TrackTable.CheckTrackTable() <> 0 THEN
			IF TrackTable.P_TrackTableCheckResult THEN
				nInitState := 50;	// Plausibility test succeeded.
			ELSE
				nInitState := 41;	// Plausibility test failed!
			END_IF
		END_IF
	41:	// In case of failed plausibility test check the creation of the above track table.
		// A Line must always begin with E_PointType.Line_Start and end with E_PointType.Line_End.
		// A Circle must always be added in the order E_PointType.Circle_Start, E_PointType.Circle_Center, E_PointType.Circle_End.
		// Check the info text for further information:
		bTrackBuildError := TRUE;
							
 					   
	50:	// Building the track	
		IF fbTrackStandard.BuildTrackExt(TrackTable) THEN
			nInitState := nInitState +1;
		END_IF
		
	51:	
		bIsDone := fbTrackStandard.P_BuildTrackExt.Done;
		bIsActive := fbTrackStandard.P_BuildTrackExt.Active;
		bIsError := fbTrackStandard.P_BuildTrackExt.Error;
		stRet := fbTrackStandard.P_BuildTrackExt;
		
		IF fbTrackStandard.P_BuildTrackExt.Done THEN
			nInitState := 100;	
		ELSIF fbTrackStandard.P_BuildTrackExt.Error THEN
	  		nInitState := nInitState +1;
		END_IF		
		
	52: // In case an error occured, check the error ID and InfoText and react accordingly:
		   bTrackBuildError := TRUE;
		 
	100: 	// Track build done
			fTrackLength := fbTrackStandard.GetLength();
			  Initialize := TRUE;
	
			
END_CASE
END_METHOD

PROPERTY P_Error : Bool
GET
P_Error := bTrackBuildError;
END_GET
END_PROPERTY

END_FUNCTION_BLOCK

// ---- Stations/FB_PuncherStation.TcPOU
FUNCTION_BLOCK FB_PuncherStation EXTENDS FB_StationBase

METHOD Clear : BOOL
	CASE nStateClear OF
		
	0:	// Enter
		Clear := FALSE;
		nStateClear := nStateClear +10;
		
	10: // Clearing all Station-Lists 
		IF SUPER^.Clear() THEN
			nStateClear := nStateClear +10;
		END_IF	
	
	20:	// Add aditional Data to be cleared here...
		nStateClear := 100;
		
		
	100: // Done
		      Clear := TRUE;
		nStateClear := 0;

	END_CASE
END_METHOD

METHOD Init : BOOL


VAR_INST
	nTestCounter	: INT;	
	
	// temp
	trackLength: LREAL;
	index: INT; 
	tempList: ARRAY[1..200] OF UDINT;
END_VAR
nTestCounter := nTestCounter +1;

CASE nStateInit OF

	0:		// Enter 
			bStationInitDone := FALSE;
			   nStateProcess := 0;
			      nStateInit := 10;
				 
			
	10:		// Init Station-Parameters				
				  nStationIndex := 1;				// Each station needs an unique index	
			 nStationTrackIndex := 1;	 			// Track on which the station resides

		
	 
	nPreviousStationIndexInputN := 1;
			  nTrackIndexInputN := 1;
	   nNextStationIndexOutputN:= 4;
	   		 nTrackIndexOutputN := 3;
			 
			 	  
			 fStationPosition_X := 600.0;			// Position of the station in X/Y coordinates
			 fStationPosition_Y := 60.0;			// Position of the station in X/Y coordinates
			  
	   fSendAwayDistanceOutputW := 500.0;			// Position on track a mover will be send to after processing 
			  fInRangeDistance  := 300.0;			// Position in front of a station from where a mover will be taken over
			  
			  nStateInit := 11;
				   
				  
	11: // Fail-safe check, just to make sure all variables have been assigned after doing copy&paste from the template
			IF        nStationIndex > 0
			AND  nStationTrackIndex > 0
			AND  nPreviousStationIndexInputN > 0
			AND  nTrackIndexInputN > 0
			AND  nNextStationIndexOutputN > 0
			AND  nTrackIndexOutputN > 0
			AND  fStationPosition_X > 0
			AND  fStationPosition_Y > 0
			//AND  fSendAwayDistanceOutputN> 0
			AND   fInRangeDistance > 0
			THEN   
				nStateInit := 20;
			END_IF
			
				   
	20:		// Calculating positions
	
			// 1. Calculating station position on track
			position.SetValuesXYC(fStationPosition_X, fStationPosition_Y, 0.0);
			trackLength := GVL.g_Tracks[nStationTrackIndex].P_TrackLength;
			//fStationPositionOnTrack := GVL.g_Tracks[nStationTrackIndex].std.GetTrackPositionAt_XY(fStationPosition_X, fStationPosition_Y);
			//fStationPositionOnTrack2 := GVL.g_Tracks[nStationTrackIndex].std.GetTrackPositionAt(position);	
			fStationPositionOnTrack := 0;  // GetTrackPositionAt only is giving rounded to 60 positions
					
			// 2. Calculating send-away position on track
			fSendAwayPositionOutputW := fStationPositionOnTrack + fSendAwayDistanceOutputW; 
			
			// The send away position must not exceed the lenght of the track!
			IF fSendAwayPositionOutputW > GVL.g_Tracks[nStationTrackIndex].P_TrackLength THEN
				fSendAwayPositionOutputW := GVL.g_Tracks[nStationTrackIndex].P_TrackLength;
			END_IF
			
			// 3. Calculating the station position in X/Y coordinates determined by the track	
            //    This is to make sure the center of the station is always located directly on the track.
			//    This value can differ from the initial fStationPosition_X, fStationPosition_Y in case they were not matching the track
			GVL.g_Tracks[nStationTrackIndex].std.GetMoverPositionAt(fStationPositionOnTrack, StationPosition);
			
			// Providing the station position to e.g. visualization	
			stStationPosition.bInit            := TRUE;
			stStationPosition.fPositionOnTrack := fStationPositionOnTrack;
			stStationPosition.nTrackId         := nStationTrackIndex;
			stStationPosition.fPosition_X	   := StationPosition.x;
			stStationPosition.fPosition_Y	   := StationPosition.y;

			nStateInit := 30;
			
			
	30:		// Clear Lists
			IF THIS^.Clear() THEN
				nStateInit := 40;	
			END_IF

	40: // create station task list 
	
	//fill hole 1-96
			
			tempList := THIS^.P_StationTaskList;

			FOR index := 1 TO 96 DO
				tempList[index] := INT_TO_UDINT(index) + 10000;
			END_FOR
			
			THIS^.P_StationTaskList := tempList;
			nStateInit := 90;
			
		
	90:		// Creating a little history of what happened in the station for debugging purpose
			fbHistoryInfo.AddEntry('Init');
	
			nStateInit := 100;
			
						
	100:	// Init done
			IF SUPER^.Init() THEN
				bStationInitDone := TRUE;	
				           Init := TRUE;
			END_IF
				
	
END_CASE
END_METHOD

METHOD Process : BOOL

VAR_INST
	
	nTaskIndex				:UINT;
	nMoverIndex				: UINT;
	com_index				:UDINT;
	nHoleIndex				: INT; 
	nMaxHoleNo				:	INT;
	RowIndex				: INT;
    ColIndex				: INT;
	
	fMoverToTrackPosition	: LREAL;
	nTrackIndex				: UINT;
	fMoverVelocity			: LREAL;
	fMoverAcceleration		: LREAL;
	fMoverJerk				: LREAL;
	
	
	nErrorId				: UDINT;
	nObjectID				: UDINT;
	nObjectType				: UDINT;		
	
	
	// Process
	nDestinationProcess		: UINT;
	nIncommingTrackOID		: UDINT;
	nNextStationIndex		: UINT;		 				
	fSendAwayPosition		: LREAL;
	nTrackindexNext			: UINT;
	bValidTask				: BOOL;
	bRotateMover			:BOOL;  
	nProcesedTask			:ST_ProcessTask;
	sProductData : ST_ProductData;
	sMoverConfiguration: REFERENCE TO ST_MoverConfiguration;
	nCmdReq					:UDINT;
	
	
	// positions 
	nextPosition : PositionXYC;
	waitPosition : PositionXYC;
	
	
	//movemets setup

	
END_VAR

VAR
	IBN_Timer:ton;
	GetP_ProcessTask: INT;
	
END_VAR

// Stop process
IF Communication.g_Com_GlobalState.IN.Stop THEN
	nStateProcess:=0;
END_IF;

// Station - Switch-Seperate
CASE nStateProcess OF 

	0:		// Enter
			IF bStationInitDone THEN
				nStateProcess := 100;
			END_IF

	
	100: 	// Waiting for Mover
			IF P_List_Switch_Input_N.P_FirstInList <> 0 THEN
				P_List_Station.AddMover(P_List_Switch_Input_N.RemoveFirstInList());
			    nStateProcess := nStateProcess +20;
				ELSE 
			//		GVL.g_Stations[GVL.PuncherStation].P_ProcessState:=ST_EStationProcessState.Empty;
			END_IF
				
			
	120: 	// Check if Mover is in range
			IF  GVL.g_Movers[nMoverIndex].std.P_SetOnTrack.TrackOID = GVL.g_Tracks[nTrackIndexInputW].std.P_OID
			AND GVL.g_Movers[nMoverIndex].std.P_SetOnTrack.SetPos   > fStationPositionOnTrack - fInRangeDistance
			AND GVL.g_Movers[nMoverIndex].P_MoverConfiguration.MoverType= TO_UINT(ST_EMoverLoadType.Wellplate)
			THEN
				nStateProcess := nStateProcess +1;
			END_IF
			
			IF GVL.g_Movers[nMoverIndex].P_MoverConfiguration.MoverType=TO_UINT(ST_EMoverLoadType.Gripper)
				THEN 
				nStateProcess := 400;				
		
			ELSIF GVL.g_Movers[nMoverIndex].P_MoverConfiguration.MoverType=TO_UINT(ST_EMoverLoadType.PipetteTips) 
				THEN 
				nStateProcess := 300;	
				
			END_IF
			
	121:	// Checking station  staus	
				CASE eProcessMode OF
				
			E_ProcessMode.None:
				;	// Nothing happens -> Process mode needs to be set!
				
			E_ProcessMode.InitRun:
				IF nStationIndex = 1 THEN
					GVL.g_Movers[nMoverIndex].P_ProductData.bInitRun := FALSE;
				//ELSE
				//	nStateProcess := 300;
				END_IF				
			
			E_ProcessMode.Production:
				nStateProcess := 200;
			
		
END_CASE

			
	200: 	// Send mover to Processing-Position
			fMoverToTrackPosition   := fStationPositionOnTrack;
			nTrackIndex        		:= nStationTrackIndex;
			fMoverVelocity     		:=    200.0;
			fMoverAcceleration 		:=  100.0;
			fMoverJerk         		:= 10_000.0;	
	
			stMoveOnTrackParameters.direction := Tc3_Mc3PlanarMotion.MC_DIRECTION.mcDirectionShortestWay;
			stMoveOnTrackParameters.gap       := 120.0;
		
			
			// Creating info text with a little history of what happened in the station for debugging purpose		
			strInfo := fbHistoryInfo.CreateStationInfo(nStationIndex, nMoverIndex, nNextStationIndex);	


			// Move on track command	
			GVL.g_Movers[nMoverIndex].std.MoveOnTrackExt( strInfo,
														GVL.g_Tracks[nTrackIndex].std,
														fMoverToTrackPosition,
														fMoverVelocity,
														fMoverAcceleration,
														fMoverJerk,
														stMoveOnTrackParameters);
			nStateProcess := nStateProcess +1;
	201: 	// Checking move command return
			IF GVL.g_Movers[nMoverIndex].std.P_MoveOnTrackExt.Done THEN
				nStateProcess := nStateProcess +9;
			ELSIF GVL.g_Movers[nMoverIndex].std.P_MoveOnTrackExt.Error THEN
				   nErrorID := GVL.g_Movers[nMoverIndex].std.P_MoveOnTrackExt.ErrorID;
				  nObjectID := GVL.g_Movers[nMoverIndex].std.P_MoveOnTrackExt.stInfo.nObjectID;
				nObjectType := GVL.g_Movers[nMoverIndex].std.P_MoveOnTrackExt.stInfo.nObjectType;
			END_IF		

	210: 
		IF NOT GVL.g_Movers[nMoverIndex].std.P_Busy THEN
			GVL.g_Movers[nMoverIndex].std.LeaveTrackInPosition( strInfo, FALSE);
			nStateProcess := nStateProcess +1;
		END_IF
		
	211:
			IF GVL.g_Movers[nMoverIndex].std.P_LeaveTrackInPosition.Done THEN
				nStateProcess := nStateProcess +9;
			ELSIF GVL.g_Movers[nMoverIndex].std.P_LeaveTrackInPosition.Error THEN
				   nErrorID := GVL.g_Movers[nMoverIndex].std.P_LeaveTrackInPosition.ErrorID;
				  nObjectID := GVL.g_Movers[nMoverIndex].std.P_LeaveTrackInPosition.stInfo.nObjectID;
				nObjectType := GVL.g_Movers[nMoverIndex].std.P_LeaveTrackInPosition.stInfo.nObjectType;
			END_IF	
		
		
	220: 	// Checking mover staus

			FOR com_index:=1 TO moverCount DO 
			IF communication.g_Com_Movers[com_index].IN.id= gvl.g_Movers[nMoverIndex].P_MoverID THEN 
			GVL.g_Movers[nMoverIndex].P_ProductData:=Communication.g_Com_Movers[com_index].ProcessData;
			END_IF
			END_FOR

 	
	
			sProductData:=GVL.g_Movers[nMoverIndex].P_ProductData;
			 IF sProductData.OK_ToProcess AND sProductData.WellplateStatus =1 THEN 
				 nStateProcess := nStateProcess +1;
				 ELSE
					 nStateProcess := 300;
					 nDestinationProcess:=3;
					 
					 
			 END_IF


	221: //check actual task is validate
	
	nProcesedTask:= GVL.g_Movers[nMoverIndex].P_ProcessTask;
	
	
		IF nProcesedTask.TaskToProcessed<>0  AND nProcesedTask.TaskToProcessed<>nProcesedTask.CurrentTask THEN 
			bValidTask:=FALSE;
			FOR  nTaskIndex:=1 TO 200 DO
				IF nProcesedTask.TaskToProcessed= nStationTaskList[nTaskIndex] THEN 
					bValidTask:=TRUE;
					nStateProcess:=nStateProcess+1;
					  RETURN;
				END_IF
			END_FOR
		
		END_IF
		
		IF bValidTask=TRUE THEN 
			nStateProcess:=nStateProcess+1;
// 		ELSE
// 			nStateProcess:=270;
		END_IF

	222: // set task to process as current task 
			nProcesedTask.CurrentTask:=nProcesedTask.TaskToProcessed;
			nProcesedTask.CurrentTaskFinished:=FALSE;
			GVL.g_Movers[nMoverIndex].P_ProcessTask:= nProcesedTask;
			nStateProcess:=nStateProcess+1;
		//	 GVL.g_Stations[GVL.PuncherStation].P_ProcessState:=ST_EStationProcessState.InProcess;
			
	223: // send mover to waiting position
			waitPosition.SetValuesXY(575,70);
	
	
		IF NOT GVL.g_Movers[nMoverIndex].std.P_Busy THEN
			stMoveToPositionOptions.useOrientation := TRUE;
			GVL.g_Movers[nMoverIndex].std.MoveToPositionExt(strInfo, waitPosition, 100, 1000, 1000, 1000, stMoveToPositionOptions);
			nStateProcess := nStateProcess +1;
		END_IF
		
	224: //check state 
			
		IF GVL.g_Movers[nMoverIndex].std.P_MoveToPositionExt.Done THEN
				nStateProcess := nStateProcess +8;
			ELSIF GVL.g_Movers[nMoverIndex].std.P_MoveToPositionExt.Error THEN
				   nErrorID := GVL.g_Movers[nMoverIndex].std.P_MoveToPositionExt.ErrorID;
				  nObjectID := GVL.g_Movers[nMoverIndex].std.P_MoveToPositionExt.stInfo.nObjectID;
				nObjectType := GVL.g_Movers[nMoverIndex].std.P_MoveToPositionExt.stInfo.nObjectType;
		END_IF

	230:// CMD to station Puncher seperate- load material 

		GVL.g_Stations[GVL.PuncherStation].P_ProcessRequest:=GVL.PuncherSeparateStation;
		
		nStateProcess:=nStateProcess+1;
	
	231:// CMD from station Puncher seperate-  material loaded
	
// 		IF  GVL.g_Stations[GVL.PuncherSeparateStation].P_ProcessState:= ST_EStationProcessState.Finished THEN 
// 			GVL.g_Stations[GVL.PuncherStation].P_ProcessRequest:=0;
// 			nStateProcess:=nStateProcess+9;
// 		END_IF

 			
	240: // calculate next position 
		bRotateMover:=FALSE;
		sMoverConfiguration REF= GVL.g_Movers[nMoverIndex].P_MoverConfiguration;
		
		nMaxHoleNo:=sMoverConfiguration.WellplateData.Columns*sMoverConfiguration.WellplateData.Row;
	
		nHoleIndex:= UDINT_TO_INT( nProcesedTask.CurrentTask MOD 10000);
		RowIndex:=0;
		ColIndex :=0; 
		
		IF 		nHoleIndex>1 THEN 
			IF  nHoleIndex< (nMaxHoleNo/2)THEN 
	
				(* row *)
				RowIndex := (nHoleIndex  / sMoverConfiguration.WellplateData.Columns)+1;
			
				(* Column *)
				ColIndex := nHoleIndex MOD sMoverConfiguration.WellplateData.Columns;
		ELSE 
			bRotateMover:=TRUE;
			nHoleIndex:=nMaxHoleNo-nHoleIndex;
			
				(* row *)
				RowIndex := (nHoleIndex  / sMoverConfiguration.WellplateData.Columns)+1;
			
				(* Column *)
				ColIndex := nHoleIndex  MOD sMoverConfiguration.WellplateData.Columns;
			
	END_IF 
END_IF
		 
    (* Calculate next position  *)
   nextPosition.x := sMoverConfiguration.WellplateData.OffsetFirstHoles_X + DINT_TO_REAL(ColIndex)* sMoverConfiguration.WellplateData.DistanceBetweenHoles_X;
   nextPosition.y := sMoverConfiguration.WellplateData.OffsetFirstHoles_Y + DINT_TO_REAL(RowIndex) * sMoverConfiguration.WellplateData.DistanceBetweenHoles_y;

nStateProcess := nStateProcess +1;



	241: // go to next position 
		
		IF NOT GVL.g_Movers[nMoverIndex].std.P_Busy THEN
			stMoveToPositionOptions.useOrientation := FALSE;
			GVL.g_Movers[nMoverIndex].std.MoveToPositionExt(strInfo, nextPosition, 100, 1000, 1000, 1000, stMoveToPositionOptions);
			nStateProcess := nStateProcess +1;
		END_IF
	242: //check state 
			IF GVL.g_Movers[nMoverIndex].std.P_MoveToPositionExt.Done THEN
				nStateProcess := nStateProcess +8;
			ELSIF GVL.g_Movers[nMoverIndex].std.P_MoveToPositionExt.Error THEN
				   nErrorID := GVL.g_Movers[nMoverIndex].std.P_MoveToPositionExt.ErrorID;
				  nObjectID := GVL.g_Movers[nMoverIndex].std.P_MoveToPositionExt.stInfo.nObjectID;
				nObjectType := GVL.g_Movers[nMoverIndex].std.P_MoveToPositionExt.stInfo.nObjectType;
			END_IF
			
	243: 
		// do rotation if needed
		IF NOT GVL.g_Movers[nMoverIndex].std.P_Busy  AND  bRotateMover THEN
			stMoveRotateOptions.additionalTurns := 0;
			stMoveRotateOptions.direction:= Tc3_Mc3PlanarMotion.MC_Direction.mcDirectionNonModulo;		
			
			GVL.g_Movers[nMoverIndex].std.MoveC(strInfo, 0.0, 100.0, 1000.0, 1000.0, 1000.0, stMoveRotateOptions);
			nStateProcess := nStateProcess +1;
			ELSE
				nStateProcess := nStateProcess +7;
		END_IF
		
	244:
			IF GVL.g_Movers[nMoverIndex].std.P_MoveC.Done THEN
				nStateProcess := nStateProcess +6;
			ELSIF GVL.g_Movers[nMoverIndex].std.P_MoveC.Error THEN
				   nErrorID := GVL.g_Movers[nMoverIndex].std.P_MoveC.ErrorID;
				  nObjectID := GVL.g_Movers[nMoverIndex].std.P_MoveC.stInfo.nObjectID;
				nObjectType := GVL.g_Movers[nMoverIndex].std.P_MoveC.stInfo.nObjectType;
			END_IF
	
 	250: // cuting 
		


	IBN_Timer(IN:=TRUE , PT:= T#3S);
			IF IBN_Timer.Q THEN 
				nStateProcess := 260;
				
			END_IF



	260:
		//update product data 
		sProductData:=GVL.g_Movers[nMoverIndex].P_ProductData;
		Communication.g_Com_Movers[nMoverIndex].ProcessData:=GVL.g_Movers[nMoverIndex].P_ProductData;
		
		
		nProcesedTask:=GVL.g_Movers[nMoverIndex].P_ProcessTask;
		nProcesedTask.CurrentTaskFinished:=TRUE;
		GVL.g_Movers[nMoverIndex].P_ProcessTask:=nProcesedTask;
		

		IF nProcesedTask.CurrentTask<>nProcesedTask.TaskToProcessed THEN  
			
			nStateProcess := nStateProcess+1;
			
		END_IF
		
	261: // check next task 
		nProcesedTask:= GVL.g_Movers[nMoverIndex].P_ProcessTask;
	
	
		IF nProcesedTask.TaskToProcessed<>0  AND nProcesedTask.TaskToProcessed<>nProcesedTask.CurrentTask THEN 
			bValidTask:=FALSE;
			FOR  nTaskIndex:=1 TO 200 DO
				IF nProcesedTask.TaskToProcessed= nStationTaskList[nTaskIndex] THEN 
					nStateProcess:=220;
					  RETURN;
				END_IF
			END_FOR
		

			IF bValidTask=TRUE THEN 
				nStateProcess:=220;
			//ELSE
// 				nStateProcess:=270;
		END_IF
		
		END_IF
		
	270: 
		// do rotation if needed
		IF NOT GVL.g_Movers[nMoverIndex].std.P_Busy THEN
			stMoveRotateOptions.additionalTurns := 0;
			stMoveRotateOptions.direction:= Tc3_Mc3PlanarMotion.MC_Direction.mcDirectionNonModulo;		
			
			GVL.g_Movers[nMoverIndex].std.MoveC(strInfo, 0.0, 100.0, 1000.0, 1000.0, 1000.0, stMoveRotateOptions);
			nStateProcess := nStateProcess +1;
		END_IF
		
	271:
			IF GVL.g_Movers[nMoverIndex].std.P_MoveC.Done THEN
				nStateProcess := nStateProcess +9;
			ELSIF GVL.g_Movers[nMoverIndex].std.P_MoveC.Error THEN
				   nErrorID := GVL.g_Movers[nMoverIndex].std.P_MoveC.ErrorID;
				  nObjectID := GVL.g_Movers[nMoverIndex].std.P_MoveC.stInfo.nObjectID;
				nObjectType := GVL.g_Movers[nMoverIndex].std.P_MoveC.stInfo.nObjectType;
			END_IF
	

	280:  // Join track
		IF NOT GVL.g_Movers[nMoverIndex].std.P_Busy THEN
			stJoinTrackOptions.useOrientation := FALSE;
			GVL.g_Movers[nMoverIndex].std.JoinTrack(strInfo, GVL.g_Tracks[nTrackIndex].std, 100, 1000, 1000, stJoinTrackOptions);
			
			nStateProcess := nStateProcess +1;
		END_IF
	281:
		IF GVL.g_Movers[nMoverIndex].std.P_JoinTrack.Done THEN
			gvl.g_Movers[nMoverIndex].P_TrackId:=nTrackIndex;
			nStateProcess := 300;
		ELSIF GVL.g_Movers[nMoverIndex].std.P_JoinTrack.Error THEN
			   nErrorID := GVL.g_Movers[nMoverIndex].std.P_JoinTrack.ErrorID;
			  nObjectID := GVL.g_Movers[nMoverIndex].std.P_JoinTrack.stInfo.nObjectID;
			nObjectType := GVL.g_Movers[nMoverIndex].std.P_JoinTrack.stInfo.nObjectType;
		END_IF	
	

	
		300: 	// Send mover to the next station
			fSendAwayPosition		:=415.95;
			fMoverToTrackPosition   := fSendAwayPosition;	
			nTrackIndex        		:= nStationTrackIndex;		
			fMoverVelocity     		:=    300.0;
			fMoverAcceleration 		:=  1_000.0;
			fMoverJerk         		:= 10_000.0;	
	
	
			stMoveOnTrackParameters.dynamicMode := MC_DYNAMICS_REDUCTION_MODE.AccelerationLimitedVelocity;
			stMoveOnTrackParameters.direction := Tc3_Mc3PlanarMotion.MC_DIRECTION.mcDirectionPositive;	
			stMoveOnTrackParameters.gap       := 120.0;

			
			// Creating info text with a little history of what happened in the station for debugging purpose		
			strInfo := fbHistoryInfo.CreateStationInfo(nStationIndex, nMoverIndex, nNextStationIndexOutputW);	
			
				
			// Move on track command	
				GVL.g_Movers[nMoverIndex].std.MoveOnTrackExt('move on track', GVL.g_Tracks[nTrackIndex].std, fMoverToTrackPosition,
 								fMoverVelocity, fMoverAcceleration , fMoverJerk, stMoveOnTrackParameters);											 
			
			nStateProcess := nStateProcess +1;
			

	301: 	// Checking move command return
			IF GVL.g_Movers[nMoverIndex].std.P_MoveOnTrackExt.Active
			OR GVL.g_Movers[nMoverIndex].std.P_MoveOnTrackExt.Done 
			THEN
				nStateProcess := nStateProcess + 9;
				
			ELSIF GVL.g_Movers[nMoverIndex].std.P_MoveOnTrackExt.Error THEN
				   nErrorID := GVL.g_Movers[nMoverIndex].std.P_MoveOnTrack.ErrorID;
				  nObjectID := GVL.g_Movers[nMoverIndex].std.P_MoveOnTrack.stInfo.nObjectID;
				nObjectType := GVL.g_Movers[nMoverIndex].std.P_MoveOnTrack.stInfo.nObjectType;
			END_IF		
		
			
	310: 	// Mover to the list of the next station
	
	
// Decide to which Station the mover has to travel to next.	
			//nDestinationProcess := 
	
						
			CASE nDestinationProcess OF
			0: // -> pipete station 
				nNextStationIndex  := nNextStationIndexOutputW ;
				nTrackindexNext    := nTrackIndexOutputW;		
		
			2: // -> buffer station 
				nNextStationIndex  := nNextStationIndexOutputN;
				nTrackindexNext    := nTrackIndexOutputN;				
	
			3: // -> User interaction
				nNextStationIndex  := nNextStationIndexOutputN;
				nTrackindexNext    := nTrackIndexOutputN;	
				nProcesedTask.CurrentTask:=50001;
				GVL.g_Movers[nMoverIndex].P_ProcessTask:=nProcesedTask;
	
			END_CASE
			
			IF nTrackindexNext > 0 THEN
				nStateProcess := 400;	
			END_IF
			
	400: 	 
		IF NOT GVL.g_Movers[nMoverIndex].std.P_Busy THEN
			GVL.g_Movers[nMoverIndex].std.LeaveTrackInPosition( strInfo, FALSE);
			nStateProcess := nStateProcess +1;
		END_IF
		
	401:
			IF GVL.g_Movers[nMoverIndex].std.P_LeaveTrackInPosition.Done THEN
				nStateProcess := nStateProcess +9;
			ELSIF GVL.g_Movers[nMoverIndex].std.P_LeaveTrackInPosition.Error THEN
				   nErrorID := GVL.g_Movers[nMoverIndex].std.P_LeaveTrackInPosition.ErrorID;
				  nObjectID := GVL.g_Movers[nMoverIndex].std.P_LeaveTrackInPosition.stInfo.nObjectID;
				nObjectType := GVL.g_Movers[nMoverIndex].std.P_LeaveTrackInPosition.stInfo.nObjectType;
			END_IF	
	402:  // Join track
		nTrackIndex:=		nTrackIndexOutputE;
		
		IF NOT GVL.g_Movers[nMoverIndex].std.P_Busy THEN
			stJoinTrackOptions.useOrientation := FALSE;
			GVL.g_Movers[nMoverIndex].std.JoinTrack(strInfo, GVL.g_Tracks[nTrackindexNext].std, 100, 1000, 1000, stJoinTrackOptions);
			
			nStateProcess := nStateProcess +1;
		END_IF
	403:
		IF GVL.g_Movers[nMoverIndex].std.P_JoinTrack.Done THEN
			gvl.g_Movers[nMoverIndex].P_TrackId:=nTrackIndex;
			nStateProcess := 300;
		ELSIF GVL.g_Movers[nMoverIndex].std.P_JoinTrack.Error THEN
			   nErrorID := GVL.g_Movers[nMoverIndex].std.P_JoinTrack.ErrorID;
			  nObjectID := GVL.g_Movers[nMoverIndex].std.P_JoinTrack.stInfo.nObjectID;
			nObjectType := GVL.g_Movers[nMoverIndex].std.P_JoinTrack.stInfo.nObjectType;
		END_IF	
	
	404:// send gripper to Puncher seperate station.
				GVL.g_Stations[nNextStationIndexOutputE].P_List_Switch_Input_S.AddMover(P_List_Station.RemoveFirstInList());

	500: //	// Done for this cycle
			//GVL.g_Stations[GVL.PuncherStation].P_ProcessState:=ST_EStationProcessState.Finished;
			nStateProcess := 100;

END_CASE
END_METHOD

END_FUNCTION_BLOCK

// ---- Stations/Base/FB_StationBase.TcPOU
FUNCTION_BLOCK FB_StationBase IMPLEMENTS I_Station


VAR
	stMoveOnTrackParameters 	: ST_MoveOnTrackOptions; 
	stMoveRotateOptions	: ST_MoveCOptions; 	
	stStationPosition	: ST_StationPosition;	
	eProcessMode		: E_ProcessMode;
	StationPosition     : PositionXYC;	
	stMoveToPositionOptions: ST_MoveToPositionOptions;
	stJoinTrackOptions: ST_JoinTrackOptions;
	stLeaveTrackOptions: ST_LeaveTrackOptions;
	
	idx  				: UDINT;
	nStateInit			: UDINT;
	nStateClear 		: UDINT;
	nStateProcess		: UDINT;
	bStationInitDone	: BOOL;	
	
	
	// Lists for Stations
	fbList_Station		: FB_List;
	fbList_InputW		: FB_List;		
	fbList_InputS		: FB_List;	
	fbList_InputE		: FB_List;		
	fbList_InputN		: FB_List;	
	
	// History info for debugging purpose
	strInfo				: STRING;	
	fbHistoryInfo		: FB_HistoryInfo;	
	
	
	nProcessRequest		: DINT;
	nProcessClearence	: DINT;
	nProcessState		: UDINT;
	
	fStationPositionOnTrack		: LREAL;	
	
	// =========================
	nStationIndex				: UINT;
	
	nPreviousStationIndexInputW : UINT;	
	nTrackIndexInputW 			: UINT;		
	nPreviousStationIndexInputS : UINT;	
	nTrackIndexInputS 			: UINT;		
	nPreviousStationIndexInputE : UINT;	
	nTrackIndexInputE 			: UINT;		
	nPreviousStationIndexInputN : UINT;	
	nTrackIndexInputN 			: UINT;		
	
	nNextStationIndexOutputW 	: UINT;	
	nTrackIndexOutputW 			: UINT;		
	nNextStationIndexOutputS 	: UINT;	
	nTrackIndexOutputS 			: UINT;		
	nNextStationIndexOutputE 	: UINT;	
	nTrackIndexOutputE 			: UINT;		
	nNextStationIndexOutputN 	: UINT;	
	nTrackIndexOutputN 			: UINT;
	
	fStationPosition_X 			: LREAL;
	fStationPosition_Y 			: LREAL;
	fInRangeDistance			: LREAL;	
	
	fSendAwayDistanceOutputW    : LREAL;	  
    fSendAwayDistanceOutputS    : LREAL;
	fSendAwayDistanceOutputE    : LREAL;	
	fSendAwayDistanceOutputN    : LREAL;
	
	fSendAwayPositionOutputW	: LREAL;
	fSendAwayPositionOutputS	: LREAL;
	fSendAwayPositionOutputE	: LREAL;
	fSendAwayPositionOutputN	: LREAL;	
	
	nStationTrackIndex			: UINT;
	nStationTaskList              :ARRAY[1..200] OF  UDINT;

	position					: PositionXYC;

	// communication data
	bComEnable			: BOOL;
	bComProcessComplete: BOOL;
	bComOK				: BOOL;
	bComNOK				: BOOL;
	bComError			: BOOL;
	nComStatusWord		: INT;
	nComErrorID			: INT;
	sComProcesedMover	: STRING(13);
	aComMoversList		: ARRAY[1..10] OF STRING(13);
	nComControlWord		: INT;
END_VAR

METHOD Clear : BOOL
VAR_INPUT
END_VAR


VAR_INST

	nStateClear : UINT;

END_VAR


	CASE nStateClear OF 
		
	0:	// Enter
		            Clear := FALSE;
		  nProcessRequest := 0;
		nProcessClearence := 0;
		    nProcessState := 0;	  
			  
		nStateClear := nStateClear +10;
		
	10: // Clear Station-List
		IF fbList_Station.ClearList() THEN
			nStateClear := nStateClear +10;	
		END_IF
		
	20: // Clear InputW-List
		IF fbList_InputW.ClearList() THEN
			nStateClear := nStateClear +10;	
		END_IF
	
	30: // Clear InputE-List
		IF fbList_InputE.ClearList() THEN
			nStateClear := nStateClear +10;	
		END_IF	
	
	40: // Clear InputS-List
		IF fbList_InputS.ClearList() THEN
			nStateClear := nStateClear +10;	
		END_IF		
	
	50: // Clear InputN-List
		IF fbList_InputN.ClearList() THEN
			nStateClear := nStateClear +10;	
		END_IF
	
	60:	nStateClear := 100;	
		
		
	100:  // Done
		nStateClear := 0;
		      Clear := TRUE;
		
	END_CASE
END_METHOD

METHOD Cycle : BOOL
VAR_INPUT
END_VAR
VAR
	nForCounter : INT;
END_VAR


VAR_INST
	
	fTestValueX	: LREAL;
	fTestValueY : LREAL;	
	
END_VAR
IF communication.RunAplicationComm AND nStationIndex > 0 AND nStationIndex <= GVL.gc_NumberStations THEN

    Communication.g_Com_Stations[nStationIndex].OUT.Enable := bComEnable;
    Communication.g_Com_Stations[nStationIndex].OUT.ProcessComplete := bComProcessComplete;
    Communication.g_Com_Stations[nStationIndex].OUT.OK := bComOK;
    Communication.g_Com_Stations[nStationIndex].OUT.NOK := bComNOK;
    Communication.g_Com_Stations[nStationIndex].OUT.Error := bComError;
    Communication.g_Com_Stations[nStationIndex].OUT.StatusWord := nComStatusWord;
    Communication.g_Com_Stations[nStationIndex].OUT.StationName := nStationIndex;
    Communication.g_Com_Stations[nStationIndex].OUT.Error_ID := nComErrorID;
    Communication.g_Com_Stations[nStationIndex].OUT.ProcesedMover := sComProcesedMover;
    Communication.g_Com_Stations[nStationIndex].OUT.MoversList := aComMoversList;

    nComControlWord := Communication.g_Com_Stations[nStationIndex].IN.ControlWord;

END_IF
END_METHOD

METHOD Init : BOOL


	  nStateInit := 0;
	nStateProcess := 0;
	 eProcessMode := E_ProcessMode.None;

	Init := TRUE;
END_METHOD

PROPERTY P_bInitDone : BOOL
GET
P_bInitDone := bStationInitDone;
END_GET
END_PROPERTY

PROPERTY P_eProcessMode : E_ProcessMode
GET
P_eProcessMode := eProcessMode;
END_GET
SET
eProcessMode := P_eProcessMode;
END_SET
END_PROPERTY

PROPERTY P_List_Station : I_List
GET
P_List_Station := fbList_Station;
END_GET
END_PROPERTY

PROPERTY P_List_Switch_Input_E : I_List
GET
P_List_Switch_Input_E := fbList_InputE;
END_GET
END_PROPERTY

{warning 'Add property implementation'}
PROPERTY P_List_Switch_Input_N : I_List
GET
P_List_Switch_Input_N := fbList_InputN;
END_GET
END_PROPERTY

PROPERTY P_List_Switch_Input_S : I_List
GET
P_List_Switch_Input_S := fbList_InputS;
END_GET
END_PROPERTY

PROPERTY P_List_Switch_Input_W : I_List
GET
P_List_Switch_Input_W := fbList_InputW;
END_GET
END_PROPERTY

PROPERTY P_nErrorCode : UDINT
GET
END_GET
END_PROPERTY

PROPERTY P_Position : ST_StationPosition
GET
P_Position := stStationPosition;
END_GET
END_PROPERTY

PROPERTY P_ProcessClearance : DINT
GET
P_ProcessClearance := nProcessClearence;
END_GET
END_PROPERTY

PROPERTY P_ProcessRequest : UDINT
GET
P_ProcessRequest := nProcessRequest;
END_GET
SET
nProcessRequest := P_ProcessRequest;
END_SET
END_PROPERTY

PROPERTY P_ProcessState : UDINT
GET
P_ProcessState := nProcessState;
END_GET
SET
nProcessState := P_ProcessState;
END_SET
END_PROPERTY

PROPERTY P_StationTaskList : array[1..200] of UDINT
GET
 P_StationTaskList := nStationTaskList;
END_GET
SET
nStationTaskList := P_StationTaskList;
END_SET
END_PROPERTY

PROPERTY P_Enable : BOOL
GET
P_Enable := bComEnable;
END_GET
SET
bComEnable := P_Enable;
END_SET
END_PROPERTY

PROPERTY P_ProcessComplete : BOOL
GET
P_ProcessComplete := bComProcessComplete;
END_GET
SET
bComProcessComplete := P_ProcessComplete;
END_SET
END_PROPERTY

PROPERTY P_OK : BOOL
GET
P_OK := bComOK;
END_GET
SET
bComOK := P_OK;
END_SET
END_PROPERTY

PROPERTY P_NOK : BOOL
GET
P_NOK := bComNOK;
END_GET
SET
bComNOK := P_NOK;
END_SET
END_PROPERTY

PROPERTY P_ComError : BOOL
GET
P_ComError := bComError;
END_GET
SET
bComError := P_ComError;
END_SET
END_PROPERTY

PROPERTY P_StatusWord : INT
GET
P_StatusWord := nComStatusWord;
END_GET
SET
nComStatusWord := P_StatusWord;
END_SET
END_PROPERTY

PROPERTY P_ComErrorID : INT
GET
P_ComErrorID := nComErrorID;
END_GET
SET
nComErrorID := P_ComErrorID;
END_SET
END_PROPERTY

PROPERTY P_ProcesedMover : STRING(13)
GET
P_ProcesedMover := sComProcesedMover;
END_GET
SET
sComProcesedMover := P_ProcesedMover;
END_SET
END_PROPERTY

PROPERTY P_MoversList : ARRAY[1..10] OF STRING(13)
GET
P_MoversList := aComMoversList;
END_GET
SET
aComMoversList := P_MoversList;
END_SET
END_PROPERTY

PROPERTY P_ControlWord : INT
GET
P_ControlWord := nComControlWord;
END_GET
SET
nComControlWord := P_ControlWord;
END_SET
END_PROPERTY

METHOD Process : BOOL
END_METHOD

END_FUNCTION_BLOCK

// ---- POUs/MAIN.TcPOU
PROGRAM MAIN
VAR
	fbXMotionUnit : FB_MotionSystem;
	nState : UDINT;
	nMemState : UDINT;
	index:UDINT;
	
	//test
	mover_idx: UINT:=1;
	
END_VAR

CASE nState OF
	0: // PELNY RESET: ustawienie nState:=0 (online) zeruje wszystkie sekwencje FB.
	   //  Startup(bReset:=TRUE) -> nStartupSequence:=0
	   //  Starting(bReset:=TRUE) -> nStartingSequence:=0 + kaskadowo Execute i MoverRecovery (patrz Starting case 0)
		fbXMotionUnit.Startup(bReset := TRUE);
		fbXMotionUnit.Starting(bReset := TRUE);
		nState := nState + 1;

	1:
		IF fbXMotionUnit.Startup(bReset := FALSE) THEN
			nState := nState + 29;
		END_IF
		
	30:
		IF fbXMotionUnit.Starting(bReset := communication.g_Com_GlobalState.IN.Reset) THEN
			nState := nState + 10;
		END_IF
		
	40: 
		fbXMotionUnit.Execute(bReset := communication.g_Com_GlobalState.IN.Reset);

		IF communication.StopApplicationComm = FALSE THEN
			
		
 			communication.RunAplicationComm:=TRUE;
		END_IF
		
	50: 
			IF fbXMotionUnit.Resetting() THEN
			nState := nMemState;
		END_IF
	
		
END_CASE


fbXMotionUnit.Cycle();

// global reset 

IF Communication.g_Com_GlobalState.IN.Reset AND nState<> 50 THEN 
	
	nMemState:=nState;
	
	nState:= 50; 
	 

END_IF



/// process parameters

Communication.g_Com_GlobalState.IN.Start:= TRUE;
//Communication.g_Com_GlobalState.IN.ProgramType:= 1; 


Communication.g_Com_Movers[mover_idx].IN.Enable:=TRUE;
Communication.g_Com_Movers[mover_idx].IN.id:= '0000lcle';
Communication.g_Com_Movers[mover_idx].IN.MoverType:=1;

Communication.g_Com_Movers[mover_idx].IN.WellplateData.Columns:=12;
Communication.g_Com_Movers[mover_idx].IN.WellplateData.Row:=9;
Communication.g_Com_Movers[mover_idx].IN.WellplateData.DistanceBetweenHoles_X:=3;
Communication.g_Com_Movers[mover_idx].IN.WellplateData.DistanceBetweenHoles_Y:=3;
Communication.g_Com_Movers[mover_idx].IN.WellplateData.OffsetFirstHoles_X:=575;
Communication.g_Com_Movers[mover_idx].IN.WellplateData.OffsetFirstHoles_Y:=70;

Communication.g_Com_Movers[mover_idx].ProcessData.OK_ToProcess:= TRUE;
Communication.g_Com_Movers[mover_idx].ProcessData.WellplateStatus:=1;

// GVL.stPayload...
// 
// 		IF GVL.ipXpu.TcIoMover(1).SetPayloadInertia(GVL.stPayload) THEN
// 			nTest := 20;
// 		END_IF
// 		
// 		IF GVL.ipXpu.TcIoMover(1).SetPayloadProductsOfInertia(GVL.stPayloadProductsOfInertia) THEN
// 			nTest := 30;
// 		END_IF

END_PROGRAM
